LIN {X 0,Y 524.002,Z 47.209,A -85,B 0,C 180,E1 -4851.516,E2 -4851.516} C_VEL
LIN {X 0,Y 524.079,Z 47.2,A -85,B 0,C 180,E1 -4854.614,E2 -4854.614} C_VEL
LIN {X 0,Y 524.108,Z 47.2,A -85,B 0,C 180,E1 -4857.695,E2 -4857.695} C_VEL
LIN {X 0,Y 524.12,Z 47.194,A -85,B 0,C 180,E1 -4860.768,E2 -4860.768} C_VEL
LIN {X 0,Y 524.069,Z 47.199,A -85,B 0,C 180,E1 -4863.075,E2 -4863.075} C_VEL
LIN {X 0,Y 524.033,Z 47.205,A -85,B 0,C 180,E1 -4866.159,E2 -4866.159} C_VEL
LIN {X 0,Y 523.99,Z 47.215,A -85,B 0,C 180,E1 -4869.262,E2 -4869.262} C_VEL
LIN {X 0,Y 524.001,Z 47.209,A -85,B 0,C 180,E1 -4871.74,E2 -4871.74} C_VEL
LIN {X 0,Y 523.991,Z 47.217,A -85,B 0,C 180,E1 -4875.053,E2 -4875.053} C_VEL
LIN {X 0,Y 523.945,Z 47.214,A -85,B 0,C 180,E1 -4877.97,E2 -4877.97} C_VEL
LIN {X 0,Y 523.97,Z 47.215,A -85,B 0,C 180,E1 -4880.41,E2 -4880.41} C_VEL
LIN {X 0,Y 523.909,Z 47.228,A -85,B 0,C 180,E1 -4882.894,E2 -4882.894} C_VEL
LIN {X 0,Y 523.933,Z 47.216,A -85,B 0,C 180,E1 -4885.42,E2 -4885.42} C_VEL
LIN {X 0,Y 523.916,Z 47.222,A -85,B 0,C 180,E1 -4888.002,E2 -4888.002} C_VEL
LIN {X 0,Y 523.943,Z 47.219,A -85,B 0,C 180,E1 -4890.855,E2 -4890.855} C_VEL
LIN {X 0,Y 523.929,Z 47.219,A -85,B 0,C 180,E1 -4893.73,E2 -4893.73} C_VEL
LIN {X 0,Y 523.897,Z 47.228,A -85,B 0,C 180,E1 -4896.401,E2 -4896.401} C_VEL
LIN {X 0,Y 523.913,Z 47.221,A -85,B 0,C 180,E1 -4899.086,E2 -4899.086} C_VEL
LIN {X 0,Y 523.908,Z 47.229,A -85,B 0,C 180,E1 -4902.124,E2 -4902.124} C_VEL
LIN {X 0,Y 523.936,Z 47.219,A -85,B 0,C 180,E1 -4905.312,E2 -4905.312} C_VEL
LIN {X 0,Y 523.886,Z 47.226,A -85,B 0,C 180,E1 -4906.905,E2 -4906.905} C_VEL
LIN {X 0,Y 523.21,Z 47.316,A -85,B 0,C 180,E1 -4907.547,E2 -4907.547} C_VEL
LIN {X 0,Y 520.363,Z 47.669,A -85,B 0,C 180,E1 -4908.589,E2 -4908.589} C_VEL
LIN {X 0,Y 517.965,Z 47.967,A -85,B 0,C 180,E1 -4909.428,E2 -4909.428} C_VEL
LIN {X 0,Y 516.94,Z 48.093,A -85,B 0,C 180,E1 -4910.075,E2 -4910.075} C_VEL
LIN {X 0,Y 516.858,Z 48.101,A -85,B 0,C 180,E1 -4910.295,E2 -4910.295} C_VEL
LIN {X 0,Y 516.847,Z 48.108,A -85,B 0,C 180,E1 -4913.348,E2 -4913.348} C_VEL
LIN {X 0,Y 516.885,Z 48.101,A -85,B 0,C 180,E1 -4916.119,E2 -4916.119} C_VEL
LIN {X 0,Y 516.927,Z 48.11,A -85,B 0,C 180,E1 -4917.452,E2 -4917.452} C_VEL
LIN {X 0,Y 517.551,Z 52.851,A -85,B 0,C 180,E1 -4918.468,E2 -4918.468} C_VEL
LIN {X 0,Y 517.344,Z 63.831,A -85,B 0,C 180,E1 -4920.702,E2 -4920.702} C_VEL
LIN {X 0,Y 519.204,Z 73.107,A -85,B 0,C 180,E1 -4920.893,E2 -4920.893} C_VEL
LIN {X 0,Y 518.694,Z 170.265,A -85,B 0,C 180,E1 -4922.268,E2 -4922.268} C_VEL
LIN {X 0,Y 518.537,Z 183.805,A -85,B 0,C 180,E1 -4922.629,E2 -4922.629} C_VEL
LIN {X 0,Y 518.349,Z 195.673,A -85,B 0,C 180,E1 -4923.095,E2 -4923.095} C_VEL
LIN {X 0,Y 518.091,Z 206.71,A -85,B 0,C 180,E1 -4923.672,E2 -4923.672} C_VEL
LIN {X 0,Y 517.742,Z 217.113,A -85,B 0,C 180,E1 -4924.363,E2 -4924.363} C_VEL
LIN {X 0,Y 517.506,Z 227.582,A -85,B 0,C 180,E1 -4925.233,E2 -4925.233} C_VEL
LIN {X 0,Y 517.214,Z 236.66,A -85,B 0,C 180,E1 -4926.156,E2 -4926.156} C_VEL
LIN {X 0,Y 516.965,Z 245.113,A -85,B 0,C 180,E1 -4927.205,E2 -4927.205} C_VEL
LIN {X 0,Y 516.759,Z 252.003,A -85,B 0,C 180,E1 -4928.247,E2 -4928.247} C_VEL
LIN {X 0,Y 516.633,Z 257.643,A -85,B 0,C 180,E1 -4929.287,E2 -4929.287} C_VEL
LIN {X 0,Y 516.506,Z 263.065,A -85,B 0,C 180,E1 -4930.527,E2 -4930.527} C_VEL
LIN {X 0,Y 516.388,Z 267.182,A -85,B 0,C 180,E1 -4931.759,E2 -4931.759} C_VEL
LIN {X 0,Y 516.329,Z 269.267,A -85,B 0,C 180,E1 -4932.576,E2 -4932.576} C_VEL
LIN {X 0,Y 516.244,Z 270.907,A -85,B 0,C 180,E1 -4933.388,E2 -4933.388} C_VEL
LIN {X 0,Y 516.251,Z 272.102,A -85,B 0,C 180,E1 -4934.201,E2 -4934.201} C_VEL
LIN {X 0,Y 516.255,Z 272.907,A -85,B 0,C 180,E1 -4935.142,E2 -4935.142} C_VEL
LIN {X 0,Y 516.244,Z 273.078,A -85,B 0,C 180,E1 -4936.619,E2 -4936.619} C_VEL
LIN {X 0,Y 516.286,Z 272.561,A -85,B 0,C 180,E1 -4937.42,E2 -4937.42} C_VEL
LIN {X 0,Y 516.347,Z 271.191,A -85,B 0,C 180,E1 -4938.522,E2 -4938.522} C_VEL
LIN {X 0,Y 516.41,Z 267.483,A -85,B 0,C 180,E1 -4940.206,E2 -4940.206} C_VEL
LIN {X 0,Y 516.456,Z 263.649,A -85,B 0,C 180,E1 -4941.391,E2 -4941.391} C_VEL
LIN {X 0,Y 516.57,Z 258.69,A -85,B 0,C 180,E1 -4942.574,E2 -4942.574} C_VEL
LIN {X 0,Y 516.716,Z 252.475,A -85,B 0,C 180,E1 -4943.754,E2 -4943.754} C_VEL
LIN {X 0,Y 516.94,Z 244.707,A -85,B 0,C 180,E1 -4944.93,E2 -4944.93} C_VEL
LIN {X 0,Y 517.232,Z 235.046,A -85,B 0,C 180,E1 -4946.105,E2 -4946.105} C_VEL
LIN {X 0,Y 517.561,Z 225.026,A -85,B 0,C 180,E1 -4947.081,E2 -4947.081} C_VEL
LIN {X 0,Y 517.844,Z 215.126,A -85,B 0,C 180,E1 -4947.861,E2 -4947.861} C_VEL
LIN {X 0,Y 518.167,Z 202.649,A -85,B 0,C 180,E1 -4948.64,E2 -4948.64} C_VEL
LIN {X 0,Y 518.388,Z 190.252,A -85,B 0,C 180,E1 -4949.223,E2 -4949.223} C_VEL
LIN {X 0,Y 518.574,Z 177.905,A -85,B 0,C 180,E1 -4949.636,E2 -4949.636} C_VEL
LIN {X 0,Y 518.709,Z 165.439,A -85,B 0,C 180,E1 -4949.903,E2 -4949.903} C_VEL
LIN {X 0,Y 519.042,Z 71.979,A -85,B 0,C 180,E1 -4951.213,E2 -4951.213} C_VEL
LIN {X 0,Y 517.23,Z 63.405,A -85,B 0,C 180,E1 -4951.411,E2 -4951.411} C_VEL
LIN {X 0,Y 517.526,Z 53.185,A -85,B 0,C 180,E1 -4953.504,E2 -4953.504} C_VEL
LIN {X 0,Y 516.921,Z 48.099,A -85,B 0,C 180,E1 -4954.582,E2 -4954.582} C_VEL
LIN {X 0,Y 517.009,Z 48.085,A -85,B 0,C 180,E1 -4957.096,E2 -4957.096} C_VEL
LIN {X 0,Y 516.95,Z 48.087,A -85,B 0,C 180,E1 -4959.39,E2 -4959.39} C_VEL
LIN {X 0,Y 516.958,Z 48.086,A -85,B 0,C 180,E1 -4961.807,E2 -4961.807} C_VEL
LIN {X 0,Y 516.951,Z 48.087,A -85,B 0,C 180,E1 -4965.147,E2 -4965.147} C_VEL
LIN {X 0,Y 516.922,Z 48.098,A -85,B 0,C 180,E1 -4968.223,E2 -4968.223} C_VEL
LIN {X 0,Y 516.918,Z 48.093,A -85,B 0,C 180,E1 -4970.701,E2 -4970.701} C_VEL
LIN {X 0,Y 516.897,Z 48.102,A -85,B 0,C 180,E1 -4974.073,E2 -4974.073} C_VEL
LIN {X 0,Y 516.931,Z 48.09,A -85,B 0,C 180,E1 -4976.658,E2 -4976.658} C_VEL
LIN {X 0,Y 516.916,Z 48.094,A -85,B 0,C 180,E1 -4979.523,E2 -4979.523} C_VEL
LIN {X 0,Y 516.901,Z 48.093,A -85,B 0,C 180,E1 -4982.543,E2 -4982.543} C_VEL
LIN {X 0,Y 516.885,Z 48.098,A -85,B 0,C 180,E1 -4985.332,E2 -4985.332} C_VEL
LIN {X 0,Y 516.885,Z 48.099,A -85,B 0,C 180,E1 -4987.943,E2 -4987.943} C_VEL
LIN {X 0,Y 516.887,Z 48.095,A -85,B 0,C 180,E1 -4990.742,E2 -4990.742} C_VEL
LIN {X 0,Y 516.887,Z 48.096,A -85,B 0,C 180,E1 -4992.831,E2 -4992.831} C_VEL
LIN {X 0,Y 516.899,Z 48.097,A -85,B 0,C 180,E1 -4995.007,E2 -4995.007} C_VEL
LIN {X 0,Y 516.917,Z 48.091,A -85,B 0,C 180,E1 -4998.399,E2 -4998.399} C_VEL
LIN {X 0,Y 516.886,Z 48.101,A -85,B 0,C 180,E1 -5001.284,E2 -5001.284} C_VEL
LIN {X 0,Y 516.875,Z 48.096,A -85,B 0,C 180,E1 -5004.22,E2 -5004.22} C_VEL
LIN {X 0,Y 516.898,Z 48.1,A -85,B 0,C 180,E1 -5007.053,E2 -5007.053} C_VEL
LIN {X 0,Y 516.896,Z 48.093,A -85,B 0,C 180,E1 -5009.796,E2 -5009.796} C_VEL
LIN {X 0,Y 516.93,Z 48.094,A -85,B 0,C 180,E1 -5012.467,E2 -5012.467} C_VEL
LIN {X 0,Y 516.914,Z 48.094,A -85,B 0,C 180,E1 -5015.072,E2 -5015.072} C_VEL
LIN {X 0,Y 516.89,Z 48.102,A -85,B 0,C 180,E1 -5018.462,E2 -5018.462} C_VEL
LIN {X 0,Y 516.904,Z 48.095,A -85,B 0,C 180,E1 -5020.955,E2 -5020.955} C_VEL
LIN {X 0,Y 516.916,Z 48.091,A -85,B 0,C 180,E1 -5023.41,E2 -5023.41} C_VEL
LIN {X 0,Y 516.897,Z 48.096,A -85,B 0,C 180,E1 -5025.833,E2 -5025.833} C_VEL
LIN {X 0,Y 516.969,Z 48.093,A -85,B 0,C 180,E1 -5028.233,E2 -5028.233} C_VEL
LIN {X 0,Y 516.968,Z 48.085,A -85,B 0,C 180,E1 -5031.399,E2 -5031.399} C_VEL
LIN {X 0,Y 517.011,Z 48.084,A -85,B 0,C 180,E1 -5033.757,E2 -5033.757} C_VEL
LIN {X 0,Y 517.084,Z 48.076,A -85,B 0,C 180,E1 -5037.663,E2 -5037.663} C_VEL
LIN {X 0,Y 517.094,Z 48.069,A -85,B 0,C 180,E1 -5040.779,E2 -5040.779} C_VEL
LIN {X 0,Y 517.012,Z 48.081,A -85,B 0,C 180,E1 -5043.117,E2 -5043.117} C_VEL
LIN {X 0,Y 517.003,Z 48.081,A -85,B 0,C 180,E1 -5046.243,E2 -5046.243} C_VEL
LIN {X 0,Y 516.949,Z 48.095,A -85,B 0,C 180,E1 -5049.389,E2 -5049.389} C_VEL
LIN {X 0,Y 516.954,Z 48.089,A -85,B 0,C 180,E1 -5051.807,E2 -5051.807} C_VEL
LIN {X 0,Y 516.947,Z 48.094,A -85,B 0,C 180,E1 -5055.146,E2 -5055.146} C_VEL
LIN {X 0,Y 516.918,Z 48.091,A -85,B 0,C 180,E1 -5058.222,E2 -5058.222} C_VEL
LIN {X 0,Y 516.914,Z 48.095,A -85,B 0,C 180,E1 -5060.701,E2 -5060.701} C_VEL
LIN {X 0,Y 516.904,Z 48.092,A -85,B 0,C 180,E1 -5064.072,E2 -5064.072} C_VEL
LIN {X 0,Y 516.906,Z 48.098,A -85,B 0,C 180,E1 -5066.659,E2 -5066.659} C_VEL
LIN {X 0,Y 516.913,Z 48.092,A -85,B 0,C 180,E1 -5069.524,E2 -5069.524} C_VEL
LIN {X 0,Y 516.897,Z 48.101,A -85,B 0,C 180,E1 -5072.543,E2 -5072.543} C_VEL
LIN {X 0,Y 516.868,Z 48.097,A -85,B 0,C 180,E1 -5075.33,E2 -5075.33} C_VEL
LIN {X 0,Y 516.882,Z 48.097,A -85,B 0,C 180,E1 -5077.943,E2 -5077.943} C_VEL
LIN {X 0,Y 516.885,Z 48.098,A -85,B 0,C 180,E1 -5080.742,E2 -5080.742} C_VEL
LIN {X 0,Y 516.884,Z 48.097,A -85,B 0,C 180,E1 -5082.831,E2 -5082.831} C_VEL
LIN {X 0,Y 516.897,Z 48.094,A -85,B 0,C 180,E1 -5085.007,E2 -5085.007} C_VEL
LIN {X 0,Y 516.915,Z 48.095,A -85,B 0,C 180,E1 -5088.399,E2 -5088.399} C_VEL
LIN {X 0,Y 516.882,Z 48.096,A -85,B 0,C 180,E1 -5091.284,E2 -5091.284} C_VEL
LIN {X 0,Y 516.873,Z 48.1,A -85,B 0,C 180,E1 -5094.22,E2 -5094.22} C_VEL
LIN {X 0,Y 516.897,Z 48.094,A -85,B 0,C 180,E1 -5097.053,E2 -5097.053} C_VEL
LIN {X 0,Y 516.89,Z 48.103,A -85,B 0,C 180,E1 -5099.796,E2 -5099.796} C_VEL
LIN {X 0,Y 516.928,Z 48.093,A -85,B 0,C 180,E1 -5102.467,E2 -5102.467} C_VEL
LIN {X 0,Y 516.966,Z 48.155,A -85,B 0,C 180,E1 -5104.536,E2 -5104.536} C_VEL
LIN {X 0,Y 518.452,Z 56.246,A -85,B 0,C 180,E1 -5105.834,E2 -5105.834} C_VEL
LIN {X 0,Y 518.155,Z 71.32,A -85,B 0,C 180,E1 -5108.099,E2 -5108.099} C_VEL
LIN {X 0,Y 517.783,Z 88.007,A -85,B 0,C 180,E1 -5110.576,E2 -5110.576} C_VEL
LIN {X 0,Y 517.364,Z 107.405,A -85,B 0,C 180,E1 -5113.425,E2 -5113.425} C_VEL
LIN {X 0,Y 517.194,Z 115.539,A -85,B 0,C 180,E1 -5114.611,E2 -5114.611} C_VEL
LIN {X 0,Y 519.007,Z 128.795,A -85,B 0,C 180,E1 -5114.864,E2 -5114.864} C_VEL
LIN {X 0,Y 518.582,Z 224.127,A -85,B 0,C 180,E1 -5116.205,E2 -5116.205} C_VEL
LIN {X 0,Y 518.303,Z 237.516,A -85,B 0,C 180,E1 -5116.548,E2 -5116.548} C_VEL
LIN {X 0,Y 518.035,Z 249.752,A -85,B 0,C 180,E1 -5117.015,E2 -5117.015} C_VEL
LIN {X 0,Y 517.755,Z 261.479,A -85,B 0,C 180,E1 -5117.617,E2 -5117.617} C_VEL
LIN {X 0,Y 517.449,Z 272.455,A -85,B 0,C 180,E1 -5118.344,E2 -5118.344} C_VEL
LIN {X 0,Y 517.167,Z 283.173,A -85,B 0,C 180,E1 -5119.23,E2 -5119.23} C_VEL
LIN {X 0,Y 516.841,Z 292.831,A -85,B 0,C 180,E1 -5120.213,E2 -5120.213} C_VEL
LIN {X 0,Y 516.653,Z 300.756,A -85,B 0,C 180,E1 -5121.197,E2 -5121.197} C_VEL
LIN {X 0,Y 516.502,Z 308.499,A -85,B 0,C 180,E1 -5122.376,E2 -5122.376} C_VEL
LIN {X 0,Y 516.353,Z 315.634,A -85,B 0,C 180,E1 -5123.749,E2 -5123.749} C_VEL
LIN {X 0,Y 516.311,Z 320.385,A -85,B 0,C 180,E1 -5124.924,E2 -5124.924} C_VEL
LIN {X 0,Y 516.369,Z 324.019,A -85,B 0,C 180,E1 -5126.098,E2 -5126.098} C_VEL
LIN {X 0,Y 516.326,Z 325.889,A -85,B 0,C 180,E1 -5126.879,E2 -5126.879} C_VEL
LIN {X 0,Y 516.266,Z 327.29,A -85,B 0,C 180,E1 -5127.659,E2 -5127.659} C_VEL
LIN {X 0,Y 516.189,Z 328.896,A -85,B 0,C 180,E1 -5129.22,E2 -5129.22} C_VEL
LIN {X 0,Y 516.194,Z 329.111,A -85,B 0,C 180,E1 -5130,E2 -5130} C_VEL
LIN {X 0,Y 516.189,Z 328.891,A -85,B 0,C 180,E1 -5130.78,E2 -5130.78} C_VEL
LIN {X 0,Y 516.266,Z 327.277,A -85,B 0,C 180,E1 -5132.34,E2 -5132.34} C_VEL
LIN {X 0,Y 516.326,Z 325.873,A -85,B 0,C 180,E1 -5133.121,E2 -5133.121} C_VEL
LIN {X 0,Y 516.311,Z 322.912,A -85,B 0,C 180,E1 -5134.293,E2 -5134.293} C_VEL
LIN {X 0,Y 516.363,Z 318.91,A -85,B 0,C 180,E1 -5135.467,E2 -5135.467} C_VEL
LIN {X 0,Y 516.405,Z 313.108,A -85,B 0,C 180,E1 -5136.771,E2 -5136.771} C_VEL
LIN {X 0,Y 516.557,Z 306.034,A -85,B 0,C 180,E1 -5138.016,E2 -5138.016} C_VEL
LIN {X 0,Y 516.723,Z 297.697,A -85,B 0,C 180,E1 -5139.196,E2 -5139.196} C_VEL
LIN {X 0,Y 516.941,Z 289.155,A -85,B 0,C 180,E1 -5140.18,E2 -5140.18} C_VEL
LIN {X 0,Y 517.281,Z 278.611,A -85,B 0,C 180,E1 -5141.163,E2 -5141.163} C_VEL
LIN {X 0,Y 517.565,Z 266.99,A -85,B 0,C 180,E1 -5142.033,E2 -5142.033} C_VEL
LIN {X 0,Y 517.952,Z 254.814,A -85,B 0,C 180,E1 -5142.738,E2 -5142.738} C_VEL
LIN {X 0,Y 518.157,Z 243.707,A -85,B 0,C 180,E1 -5143.231,E2 -5143.231} C_VEL
LIN {X 0,Y 518.419,Z 230.576,A -85,B 0,C 180,E1 -5143.648,E2 -5143.648} C_VEL
LIN {X 0,Y 518.65,Z 218.043,A -85,B 0,C 180,E1 -5143.892,E2 -5143.892} C_VEL
LIN {X 0,Y 518.952,Z 128.16,A -85,B 0,C 180,E1 -5145.145,E2 -5145.145} C_VEL
LIN {X 0,Y 517.214,Z 115.433,A -85,B 0,C 180,E1 -5145.384,E2 -5145.384} C_VEL
LIN {X 0,Y 517.715,Z 92.05,A -85,B 0,C 180,E1 -5148.808,E2 -5148.808} C_VEL
LIN {X 0,Y 518.116,Z 72.687,A -85,B 0,C 180,E1 -5151.693,E2 -5151.693} C_VEL
LIN {X 0,Y 518.514,Z 56.387,A -85,B 0,C 180,E1 -5154.161,E2 -5154.161} C_VEL
LIN {X 0,Y 516.943,Z 48.093,A -85,B 0,C 180,E1 -5155.545,E2 -5155.545} C_VEL
LIN {X 0,Y 516.92,Z 48.099,A -85,B 0,C 180,E1 -5158.415,E2 -5158.415} C_VEL
LIN {X 0,Y 516.889,Z 48.098,A -85,B 0,C 180,E1 -5161.109,E2 -5161.109} C_VEL
LIN {X 0,Y 516.891,Z 48.103,A -85,B 0,C 180,E1 -5163.963,E2 -5163.963} C_VEL
LIN {X 0,Y 516.883,Z 48.097,A -85,B 0,C 180,E1 -5166.745,E2 -5166.745} C_VEL
LIN {X 0,Y 516.881,Z 48.103,A -85,B 0,C 180,E1 -5169.721,E2 -5169.721} C_VEL
LIN {X 0,Y 516.91,Z 48.1,A -85,B 0,C 180,E1 -5171.775,E2 -5171.775} C_VEL
LIN {X 0,Y 516.893,Z 48.094,A -85,B 0,C 180,E1 -5175.007,E2 -5175.007} C_VEL
LIN {X 0,Y 516.921,Z 48.091,A -85,B 0,C 180,E1 -5178.397,E2 -5178.397} C_VEL
LIN {X 0,Y 516.885,Z 48.103,A -85,B 0,C 180,E1 -5181.284,E2 -5181.284} C_VEL
LIN {X 0,Y 516.89,Z 48.095,A -85,B 0,C 180,E1 -5184.221,E2 -5184.221} C_VEL
LIN {X 0,Y 516.894,Z 48.101,A -85,B 0,C 180,E1 -5187.053,E2 -5187.053} C_VEL
LIN {X 0,Y 516.89,Z 48.094,A -85,B 0,C 180,E1 -5189.796,E2 -5189.796} C_VEL
LIN {X 0,Y 516.926,Z 48.093,A -85,B 0,C 180,E1 -5192.467,E2 -5192.467} C_VEL
LIN {X 0,Y 516.909,Z 48.097,A -85,B 0,C 180,E1 -5195.072,E2 -5195.072} C_VEL
LIN {X 0,Y 516.867,Z 48.094,A -85,B 0,C 180,E1 -5197.621,E2 -5197.621} C_VEL
LIN {X 0,Y 516.93,Z 48.092,A -85,B 0,C 180,E1 -5200.13,E2 -5200.13} C_VEL
LIN {X 0,Y 516.927,Z 48.095,A -85,B 0,C 180,E1 -5202.596,E2 -5202.596} C_VEL
LIN {X 0,Y 516.94,Z 48.089,A -85,B 0,C 180,E1 -5205.03,E2 -5205.03} C_VEL
LIN {X 0,Y 516.963,Z 48.09,A -85,B 0,C 180,E1 -5208.234,E2 -5208.234} C_VEL
LIN {X 0,Y 516.967,Z 48.085,A -85,B 0,C 180,E1 -5211.4,E2 -5211.4} C_VEL
LIN {X 0,Y 517.007,Z 48.083,A -85,B 0,C 180,E1 -5213.757,E2 -5213.757} C_VEL
LIN {X 0,Y 517.08,Z 48.075,A -85,B 0,C 180,E1 -5217.663,E2 -5217.663} C_VEL
LIN {X 0,Y 517.091,Z 48.07,A -85,B 0,C 180,E1 -5220.779,E2 -5220.779} C_VEL
LIN {X 0,Y 517.009,Z 48.079,A -85,B 0,C 180,E1 -5223.117,E2 -5223.117} C_VEL
LIN {X 0,Y 516.999,Z 48.081,A -85,B 0,C 180,E1 -5226.244,E2 -5226.244} C_VEL
LIN {X 0,Y 516.946,Z 48.094,A -85,B 0,C 180,E1 -5229.39,E2 -5229.39} C_VEL
LIN {X 0,Y 516.95,Z 48.087,A -85,B 0,C 180,E1 -5231.807,E2 -5231.807} C_VEL
LIN {X 0,Y 516.943,Z 48.096,A -85,B 0,C 180,E1 -5235.147,E2 -5235.147} C_VEL
LIN {X 0,Y 516.914,Z 48.09,A -85,B 0,C 180,E1 -5238.223,E2 -5238.223} C_VEL
LIN {X 0,Y 516.911,Z 48.099,A -85,B 0,C 180,E1 -5240.702,E2 -5240.702} C_VEL
LIN {X 0,Y 516.9,Z 48.095,A -85,B 0,C 180,E1 -5244.073,E2 -5244.073} C_VEL
LIN {X 0,Y 516.896,Z 48.101,A -85,B 0,C 180,E1 -5246.66,E2 -5246.66} C_VEL
LIN {X 0,Y 516.909,Z 48.091,A -85,B 0,C 180,E1 -5249.524,E2 -5249.524} C_VEL
LIN {X 0,Y 516.893,Z 48.1,A -85,B 0,C 180,E1 -5252.544,E2 -5252.544} C_VEL
LIN {X 0,Y 516.861,Z 48.097,A -85,B 0,C 180,E1 -5255.329,E2 -5255.329} C_VEL
LIN {X 0,Y 516.878,Z 48.103,A -85,B 0,C 180,E1 -5257.943,E2 -5257.943} C_VEL
LIN {X 0,Y 516.853,Z 48.097,A -85,B 0,C 180,E1 -5260.745,E2 -5260.745} C_VEL
LIN {X 0,Y 516.88,Z 48.104,A -85,B 0,C 180,E1 -5263.904,E2 -5263.904} C_VEL
LIN {X 0,Y 516.84,Z 48.104,A -85,B 0,C 180,E1 -5266.906,E2 -5266.906} C_VEL
LIN {X 0,Y 516.861,Z 48.107,A -85,B 0,C 180,E1 -5269.594,E2 -5269.594} C_VEL
LIN {X 0,Y 516.858,Z 48.101,A -85,B 0,C 180,E1 -5270.295,E2 -5270.295} C_VEL
LIN {X 0,Y 516.196,Z 48.184,A -85,B 0,C 180,E1 -5270.945,E2 -5270.945} C_VEL
LIN {X 0,Y 513.345,Z 48.545,A -85,B 0,C 180,E1 -5272,E2 -5272} C_VEL
LIN {X 0,Y 510.929,Z 48.849,A -85,B 0,C 180,E1 -5272.851,E2 -5272.851} C_VEL
LIN {X 0,Y 509.888,Z 48.976,A -85,B 0,C 180,E1 -5273.507,E2 -5273.507} C_VEL
LIN {X 0,Y 509.802,Z 48.985,A -85,B 0,C 180,E1 -5273.73,E2 -5273.73} C_VEL
LIN {X 0,Y 509.849,Z 48.978,A -85,B 0,C 180,E1 -5276.539,E2 -5276.539} C_VEL
LIN {X 0,Y 509.91,Z 49.086,A -85,B 0,C 180,E1 -5277.322,E2 -5277.322} C_VEL
LIN {X 0,Y 510.594,Z 54.905,A -85,B 0,C 180,E1 -5278.583,E2 -5278.583} C_VEL
LIN {X 0,Y 510.368,Z 64.136,A -85,B 0,C 180,E1 -5280.478,E2 -5280.478} C_VEL
LIN {X 0,Y 512.376,Z 74.317,A -85,B 0,C 180,E1 -5280.692,E2 -5280.692} C_VEL
LIN {X 0,Y 511.822,Z 170.404,A -85,B 0,C 180,E1 -5282.071,E2 -5282.071} C_VEL
LIN {X 0,Y 511.635,Z 184.046,A -85,B 0,C 180,E1 -5282.436,E2 -5282.436} C_VEL
LIN {X 0,Y 511.442,Z 196.255,A -85,B 0,C 180,E1 -5282.923,E2 -5282.923} C_VEL
LIN {X 0,Y 511.12,Z 208.288,A -85,B 0,C 180,E1 -5283.574,E2 -5283.574} C_VEL
LIN {X 0,Y 510.759,Z 218.975,A -85,B 0,C 180,E1 -5284.315,E2 -5284.315} C_VEL
LIN {X 0,Y 510.464,Z 229.831,A -85,B 0,C 180,E1 -5285.257,E2 -5285.257} C_VEL
LIN {X 0,Y 510.17,Z 238.963,A -85,B 0,C 180,E1 -5286.238,E2 -5286.238} C_VEL
LIN {X 0,Y 509.869,Z 248.021,A -85,B 0,C 180,E1 -5287.448,E2 -5287.448} C_VEL
LIN {X 0,Y 509.653,Z 254.798,A -85,B 0,C 180,E1 -5288.566,E2 -5288.566} C_VEL
LIN {X 0,Y 509.519,Z 260.942,A -85,B 0,C 180,E1 -5289.829,E2 -5289.829} C_VEL
LIN {X 0,Y 509.36,Z 265.677,A -85,B 0,C 180,E1 -5291.08,E2 -5291.08} C_VEL
LIN {X 0,Y 509.273,Z 269.205,A -85,B 0,C 180,E1 -5292.326,E2 -5292.326} C_VEL
LIN {X 0,Y 509.196,Z 270.929,A -85,B 0,C 180,E1 -5293.152,E2 -5293.152} C_VEL
LIN {X 0,Y 509.178,Z 272.225,A -85,B 0,C 180,E1 -5293.976,E2 -5293.976} C_VEL
LIN {X 0,Y 509.176,Z 273.25,A -85,B 0,C 180,E1 -5295.06,E2 -5295.06} C_VEL
LIN {X 0,Y 509.149,Z 273.502,A -85,B 0,C 180,E1 -5296.429,E2 -5296.429} C_VEL
LIN {X 0,Y 509.189,Z 273.11,A -85,B 0,C 180,E1 -5297.242,E2 -5297.242} C_VEL
LIN {X 0,Y 509.257,Z 271.687,A -85,B 0,C 180,E1 -5298.477,E2 -5298.477} C_VEL
LIN {X 0,Y 509.313,Z 268.385,A -85,B 0,C 180,E1 -5300.068,E2 -5300.068} C_VEL
LIN {X 0,Y 509.387,Z 264.72,A -85,B 0,C 180,E1 -5301.271,E2 -5301.271} C_VEL
LIN {X 0,Y 509.495,Z 259.945,A -85,B 0,C 180,E1 -5302.47,E2 -5302.47} C_VEL
LIN {X 0,Y 509.672,Z 252.821,A -85,B 0,C 180,E1 -5303.866,E2 -5303.866} C_VEL
LIN {X 0,Y 509.923,Z 245.037,A -85,B 0,C 180,E1 -5305.059,E2 -5305.059} C_VEL
LIN {X 0,Y 510.246,Z 235.36,A -85,B 0,C 180,E1 -5306.249,E2 -5306.249} C_VEL
LIN {X 0,Y 510.595,Z 225.316,A -85,B 0,C 180,E1 -5307.239,E2 -5307.239} C_VEL
LIN {X 0,Y 510.915,Z 215.385,A -85,B 0,C 180,E1 -5308.03,E2 -5308.03} C_VEL
LIN {X 0,Y 511.224,Z 204.606,A -85,B 0,C 180,E1 -5308.72,E2 -5308.72} C_VEL
LIN {X 0,Y 511.454,Z 192.762,A -85,B 0,C 180,E1 -5309.311,E2 -5309.311} C_VEL
LIN {X 0,Y 511.676,Z 180.616,A -85,B 0,C 180,E1 -5309.754,E2 -5309.754} C_VEL
LIN {X 0,Y 511.819,Z 168.222,A -85,B 0,C 180,E1 -5310.049,E2 -5310.049} C_VEL
LIN {X 0,Y 512.176,Z 72.822,A -85,B 0,C 180,E1 -5311.41,E2 -5311.41} C_VEL
LIN {X 0,Y 510.272,Z 63.821,A -85,B 0,C 180,E1 -5311.603,E2 -5311.603} C_VEL
LIN {X 0,Y 510.462,Z 52.48,A -85,B 0,C 180,E1 -5313.948,E2 -5313.948} C_VEL
LIN {X 0,Y 509.906,Z 48.973,A -85,B 0,C 180,E1 -5314.744,E2 -5314.744} C_VEL
LIN {X 0,Y 509.981,Z 48.96,A -85,B 0,C 180,E1 -5317.145,E2 -5317.145} C_VEL
LIN {X 0,Y 509.861,Z 48.975,A -85,B 0,C 180,E1 -5320.323,E2 -5320.323} C_VEL
LIN {X 0,Y 509.883,Z 48.972,A -85,B 0,C 180,E1 -5322.741,E2 -5322.741} C_VEL
LIN {X 0,Y 509.9,Z 48.965,A -85,B 0,C 180,E1 -5325.242,E2 -5325.242} C_VEL
LIN {X 0,Y 509.867,Z 48.975,A -85,B 0,C 180,E1 -5328.484,E2 -5328.484} C_VEL
LIN {X 0,Y 509.856,Z 48.971,A -85,B 0,C 180,E1 -5331.002,E2 -5331.002} C_VEL
LIN {X 0,Y 509.828,Z 48.976,A -85,B 0,C 180,E1 -5333.564,E2 -5333.564} C_VEL
LIN {X 0,Y 509.917,Z 48.966,A -85,B 0,C 180,E1 -5336.378,E2 -5336.378} C_VEL
LIN {X 0,Y 509.878,Z 48.968,A -85,B 0,C 180,E1 -5338.844,E2 -5338.844} C_VEL
LIN {X 0,Y 509.826,Z 48.979,A -85,B 0,C 180,E1 -5341.59,E2 -5341.59} C_VEL
LIN {X 0,Y 509.858,Z 48.971,A -85,B 0,C 180,E1 -5344.413,E2 -5344.413} C_VEL
LIN {X 0,Y 509.823,Z 48.979,A -85,B 0,C 180,E1 -5347.341,E2 -5347.341} C_VEL
LIN {X 0,Y 509.843,Z 48.972,A -85,B 0,C 180,E1 -5350.382,E2 -5350.382} C_VEL
LIN {X 0,Y 509.827,Z 48.977,A -85,B 0,C 180,E1 -5353.062,E2 -5353.062} C_VEL
LIN {X 0,Y 509.826,Z 48.977,A -85,B 0,C 180,E1 -5355.793,E2 -5355.793} C_VEL
LIN {X 0,Y 509.859,Z 48.971,A -85,B 0,C 180,E1 -5358.574,E2 -5358.574} C_VEL
LIN {X 0,Y 509.855,Z 48.972,A -85,B 0,C 180,E1 -5361.786,E2 -5361.786} C_VEL
LIN {X 0,Y 509.835,Z 48.976,A -85,B 0,C 180,E1 -5364.622,E2 -5364.622} C_VEL
LIN {X 0,Y 509.865,Z 48.971,A -85,B 0,C 180,E1 -5367.481,E2 -5367.481} C_VEL
LIN {X 0,Y 509.862,Z 48.971,A -85,B 0,C 180,E1 -5370.273,E2 -5370.273} C_VEL
LIN {X 0,Y 509.887,Z 48.972,A -85,B 0,C 180,E1 -5372.944,E2 -5372.944} C_VEL
LIN {X 0,Y 509.874,Z 48.968,A -85,B 0,C 180,E1 -5375.574,E2 -5375.574} C_VEL
LIN {X 0,Y 509.854,Z 48.973,A -85,B 0,C 180,E1 -5378.998,E2 -5378.998} C_VEL
LIN {X 0,Y 509.885,Z 48.97,A -85,B 0,C 180,E1 -5382.001,E2 -5382.001} C_VEL
LIN {X 0,Y 509.914,Z 48.965,A -85,B 0,C 180,E1 -5384.819,E2 -5384.819} C_VEL
LIN {X 0,Y 509.904,Z 48.972,A -85,B 0,C 180,E1 -5388.124,E2 -5388.124} C_VEL
LIN {X 0,Y 509.914,Z 48.963,A -85,B 0,C 180,E1 -5391.28,E2 -5391.28} C_VEL
LIN {X 0,Y 509.962,Z 48.961,A -85,B 0,C 180,E1 -5393.67,E2 -5393.67} C_VEL
LIN {X 0,Y 510.055,Z 48.951,A -85,B 0,C 180,E1 -5397.631,E2 -5397.631} C_VEL
LIN {X 0,Y 510.065,Z 48.944,A -85,B 0,C 180,E1 -5400.789,E2 -5400.789} C_VEL
LIN {X 0,Y 509.954,Z 48.96,A -85,B 0,C 180,E1 -5403.16,E2 -5403.16} C_VEL
LIN {X 0,Y 509.954,Z 48.959,A -85,B 0,C 180,E1 -5406.33,E2 -5406.33} C_VEL
LIN {X 0,Y 509.89,Z 48.974,A -85,B 0,C 180,E1 -5409.52,E2 -5409.52} C_VEL
LIN {X 0,Y 509.907,Z 48.966,A -85,B 0,C 180,E1 -5411.931,E2 -5411.931} C_VEL
LIN {X 0,Y 509.896,Z 48.974,A -85,B 0,C 180,E1 -5415.242,E2 -5415.242} C_VEL
LIN {X 0,Y 509.869,Z 48.969,A -85,B 0,C 180,E1 -5417.993,E2 -5417.993} C_VEL
LIN {X 0,Y 509.888,Z 48.967,A -85,B 0,C 180,E1 -5420.401,E2 -5420.401} C_VEL
LIN {X 0,Y 509.831,Z 48.975,A -85,B 0,C 180,E1 -5423.563,E2 -5423.563} C_VEL
LIN {X 0,Y 509.888,Z 48.969,A -85,B 0,C 180,E1 -5426.372,E2 -5426.372} C_VEL
LIN {X 0,Y 509.874,Z 48.976,A -85,B 0,C 180,E1 -5428.844,E2 -5428.844} C_VEL
LIN {X 0,Y 509.821,Z 48.975,A -85,B 0,C 180,E1 -5431.59,E2 -5431.59} C_VEL
LIN {X 0,Y 509.849,Z 48.977,A -85,B 0,C 180,E1 -5434.414,E2 -5434.414} C_VEL
LIN {X 0,Y 509.818,Z 48.975,A -85,B 0,C 180,E1 -5437.341,E2 -5437.341} C_VEL
LIN {X 0,Y 509.84,Z 48.981,A -85,B 0,C 180,E1 -5440.382,E2 -5440.382} C_VEL
LIN {X 0,Y 509.824,Z 48.975,A -85,B 0,C 180,E1 -5443.062,E2 -5443.062} C_VEL
LIN {X 0,Y 509.824,Z 48.978,A -85,B 0,C 180,E1 -5445.793,E2 -5445.793} C_VEL
LIN {X 0,Y 509.857,Z 48.972,A -85,B 0,C 180,E1 -5448.574,E2 -5448.574} C_VEL
LIN {X 0,Y 509.852,Z 48.977,A -85,B 0,C 180,E1 -5451.787,E2 -5451.787} C_VEL
LIN {X 0,Y 509.832,Z 48.974,A -85,B 0,C 180,E1 -5454.622,E2 -5454.622} C_VEL
LIN {X 0,Y 509.863,Z 48.974,A -85,B 0,C 180,E1 -5457.481,E2 -5457.481} C_VEL
LIN {X 0,Y 509.861,Z 48.976,A -85,B 0,C 180,E1 -5460.274,E2 -5460.274} C_VEL
LIN {X 0,Y 509.886,Z 48.972,A -85,B 0,C 180,E1 -5462.944,E2 -5462.944} C_VEL
LIN {X 0,Y 509.93,Z 49.078,A -85,B 0,C 180,E1 -5464.379,E2 -5464.379} C_VEL
LIN {X 0,Y 511.559,Z 58.313,A -85,B 0,C 180,E1 -5465.875,E2 -5465.875} C_VEL
LIN {X 0,Y 511.097,Z 77.853,A -85,B 0,C 180,E1 -5468.841,E2 -5468.841} C_VEL
LIN {X 0,Y 510.566,Z 100.441,A -85,B 0,C 180,E1 -5472.219,E2 -5472.219} C_VEL
LIN {X 0,Y 510.178,Z 115.221,A -85,B 0,C 180,E1 -5474.406,E2 -5474.406} C_VEL
LIN {X 0,Y 512.136,Z 129.771,A -85,B 0,C 180,E1 -5474.678,E2 -5474.678} C_VEL
LIN {X 0,Y 511.675,Z 224.809,A -85,B 0,C 180,E1 -5476.041,E2 -5476.041} C_VEL
LIN {X 0,Y 511.363,Z 237.843,A -85,B 0,C 180,E1 -5476.387,E2 -5476.387} C_VEL
LIN {X 0,Y 511.076,Z 250.467,A -85,B 0,C 180,E1 -5476.885,E2 -5476.885} C_VEL
LIN {X 0,Y 510.748,Z 262.481,A -85,B 0,C 180,E1 -5477.533,E2 -5477.533} C_VEL
LIN {X 0,Y 510.432,Z 273.362,A -85,B 0,C 180,E1 -5478.282,E2 -5478.282} C_VEL
LIN {X 0,Y 510.122,Z 283.86,A -85,B 0,C 180,E1 -5479.18,E2 -5479.18} C_VEL
LIN {X 0,Y 509.804,Z 292.443,A -85,B 0,C 180,E1 -5480.077,E2 -5480.077} C_VEL
LIN {X 0,Y 509.6,Z 300.369,A -85,B 0,C 180,E1 -5481.074,E2 -5481.074} C_VEL
LIN {X 0,Y 509.415,Z 308.113,A -85,B 0,C 180,E1 -5482.269,E2 -5482.269} C_VEL
LIN {X 0,Y 509.259,Z 315.249,A -85,B 0,C 180,E1 -5483.661,E2 -5483.661} C_VEL
LIN {X 0,Y 509.239,Z 320.002,A -85,B 0,C 180,E1 -5484.853,E2 -5484.853} C_VEL
LIN {X 0,Y 509.275,Z 323.635,A -85,B 0,C 180,E1 -5486.043,E2 -5486.043} C_VEL
LIN {X 0,Y 509.241,Z 325.506,A -85,B 0,C 180,E1 -5486.835,E2 -5486.835} C_VEL
LIN {X 0,Y 509.196,Z 326.908,A -85,B 0,C 180,E1 -5487.627,E2 -5487.627} C_VEL
LIN {X 0,Y 509.101,Z 328.512,A -85,B 0,C 180,E1 -5489.209,E2 -5489.209} C_VEL
LIN {X 0,Y 509.105,Z 328.727,A -85,B 0,C 180,E1 -5490,E2 -5490} C_VEL
LIN {X 0,Y 509.12,Z 327.893,A -85,B 0,C 180,E1 -5491.582,E2 -5491.582} C_VEL
LIN {X 0,Y 509.196,Z 326.892,A -85,B 0,C 180,E1 -5492.373,E2 -5492.373} C_VEL
LIN {X 0,Y 509.241,Z 325.485,A -85,B 0,C 180,E1 -5493.164,E2 -5493.164} C_VEL
LIN {X 0,Y 509.204,Z 322.522,A -85,B 0,C 180,E1 -5494.353,E2 -5494.353} C_VEL
LIN {X 0,Y 509.272,Z 318.518,A -85,B 0,C 180,E1 -5495.543,E2 -5495.543} C_VEL
LIN {X 0,Y 509.329,Z 312.462,A -85,B 0,C 180,E1 -5496.914,E2 -5496.914} C_VEL
LIN {X 0,Y 509.476,Z 305.636,A -85,B 0,C 180,E1 -5498.128,E2 -5498.128} C_VEL
LIN {X 0,Y 509.68,Z 297.298,A -85,B 0,C 180,E1 -5499.324,E2 -5499.324} C_VEL
LIN {X 0,Y 509.926,Z 288.754,A -85,B 0,C 180,E1 -5500.321,E2 -5500.321} C_VEL
LIN {X 0,Y 510.291,Z 278.212,A -85,B 0,C 180,E1 -5501.318,E2 -5501.318} C_VEL
LIN {X 0,Y 510.565,Z 267.349,A -85,B 0,C 180,E1 -5502.148,E2 -5502.148} C_VEL
LIN {X 0,Y 510.955,Z 256.366,A -85,B 0,C 180,E1 -5502.814,E2 -5502.814} C_VEL
LIN {X 0,Y 511.207,Z 244.634,A -85,B 0,C 180,E1 -5503.364,E2 -5503.364} C_VEL
LIN {X 0,Y 511.5,Z 231.133,A -85,B 0,C 180,E1 -5503.811,E2 -5503.811} C_VEL
LIN {X 0,Y 511.774,Z 217.732,A -85,B 0,C 180,E1 -5504.083,E2 -5504.083} C_VEL
LIN {X 0,Y 511.993,Z 128.102,A -85,B 0,C 180,E1 -5505.355,E2 -5505.355} C_VEL
LIN {X 0,Y 510.187,Z 115.008,A -85,B 0,C 180,E1 -5505.608,E2 -5505.608} C_VEL
LIN {X 0,Y 510.724,Z 93.109,A -85,B 0,C 180,E1 -5508.867,E2 -5508.867} C_VEL
LIN {X 0,Y 511.168,Z 73.779,A -85,B 0,C 180,E1 -5511.791,E2 -5511.791} C_VEL
LIN {X 0,Y 511.643,Z 58.613,A -85,B 0,C 180,E1 -5514.12,E2 -5514.12} C_VEL
LIN {X 0,Y 509.919,Z 48.968,A -85,B 0,C 180,E1 -5515.731,E2 -5515.731} C_VEL
LIN {X 0,Y 509.877,Z 48.974,A -85,B 0,C 180,E1 -5518.844,E2 -5518.844} C_VEL
LIN {X 0,Y 509.82,Z 48.98,A -85,B 0,C 180,E1 -5521.59,E2 -5521.59} C_VEL
LIN {X 0,Y 509.845,Z 48.976,A -85,B 0,C 180,E1 -5524.413,E2 -5524.413} C_VEL
LIN {X 0,Y 509.819,Z 48.978,A -85,B 0,C 180,E1 -5527.34,E2 -5527.34} C_VEL
LIN {X 0,Y 509.837,Z 48.976,A -85,B 0,C 180,E1 -5530.382,E2 -5530.382} C_VEL
LIN {X 0,Y 509.822,Z 48.977,A -85,B 0,C 180,E1 -5533.062,E2 -5533.062} C_VEL
LIN {X 0,Y 509.821,Z 48.977,A -85,B 0,C 180,E1 -5535.793,E2 -5535.793} C_VEL
LIN {X 0,Y 509.864,Z 48.97,A -85,B 0,C 180,E1 -5538.575,E2 -5538.575} C_VEL
LIN {X 0,Y 509.851,Z 48.972,A -85,B 0,C 180,E1 -5541.786,E2 -5541.786} C_VEL
LIN {X 0,Y 509.845,Z 48.974,A -85,B 0,C 180,E1 -5544.623,E2 -5544.623} C_VEL
LIN {X 0,Y 509.861,Z 48.974,A -85,B 0,C 180,E1 -5547.481,E2 -5547.481} C_VEL
LIN {X 0,Y 509.856,Z 48.971,A -85,B 0,C 180,E1 -5550.273,E2 -5550.273} C_VEL
LIN {X 0,Y 509.883,Z 48.972,A -85,B 0,C 180,E1 -5552.944,E2 -5552.944} C_VEL
LIN {X 0,Y 509.868,Z 48.97,A -85,B 0,C 180,E1 -5555.574,E2 -5555.574} C_VEL
LIN {X 0,Y 509.82,Z 48.974,A -85,B 0,C 180,E1 -5558.149,E2 -5558.149} C_VEL
LIN {X 0,Y 509.862,Z 48.975,A -85,B 0,C 180,E1 -5560.682,E2 -5560.682} C_VEL
LIN {X 0,Y 509.882,Z 48.967,A -85,B 0,C 180,E1 -5563.175,E2 -5563.175} C_VEL
LIN {X 0,Y 509.862,Z 48.971,A -85,B 0,C 180,E1 -5565.634,E2 -5565.634} C_VEL
LIN {X 0,Y 509.912,Z 48.965,A -85,B 0,C 180,E1 -5568.875,E2 -5568.875} C_VEL
LIN {X 0,Y 509.949,Z 48.963,A -85,B 0,C 180,E1 -5572.079,E2 -5572.079} C_VEL
LIN {X 0,Y 509.979,Z 48.958,A -85,B 0,C 180,E1 -5574.464,E2 -5574.464} C_VEL
LIN {X 0,Y 510.051,Z 48.95,A -85,B 0,C 180,E1 -5577.631,E2 -5577.631} C_VEL
LIN {X 0,Y 510.061,Z 48.945,A -85,B 0,C 180,E1 -5580.79,E2 -5580.79} C_VEL
LIN {X 0,Y 509.951,Z 48.958,A -85,B 0,C 180,E1 -5583.16,E2 -5583.16} C_VEL
LIN {X 0,Y 509.95,Z 48.959,A -85,B 0,C 180,E1 -5586.33,E2 -5586.33} C_VEL
LIN {X 0,Y 509.887,Z 48.973,A -85,B 0,C 180,E1 -5589.521,E2 -5589.521} C_VEL
LIN {X 0,Y 509.902,Z 48.964,A -85,B 0,C 180,E1 -5591.932,E2 -5591.932} C_VEL
LIN {X 0,Y 509.892,Z 48.973,A -85,B 0,C 180,E1 -5595.242,E2 -5595.242} C_VEL
LIN {X 0,Y 509.865,Z 48.967,A -85,B 0,C 180,E1 -5597.994,E2 -5597.994} C_VEL
LIN {X 0,Y 509.885,Z 48.97,A -85,B 0,C 180,E1 -5600.402,E2 -5600.402} C_VEL
LIN {X 0,Y 509.827,Z 48.975,A -85,B 0,C 180,E1 -5603.564,E2 -5603.564} C_VEL
LIN {X 0,Y 509.877,Z 48.971,A -85,B 0,C 180,E1 -5606.371,E2 -5606.371} C_VEL
LIN {X 0,Y 509.857,Z 48.97,A -85,B 0,C 180,E1 -5609.727,E2 -5609.727} C_VEL
LIN {X 0,Y 509.866,Z 48.973,A -85,B 0,C 180,E1 -5612.773,E2 -5612.773} C_VEL
LIN {X 0,Y 509.821,Z 48.975,A -85,B 0,C 180,E1 -5615.578,E2 -5615.578} C_VEL
LIN {X 0,Y 509.848,Z 48.979,A -85,B 0,C 180,E1 -5618.339,E2 -5618.339} C_VEL
LIN {X 0,Y 509.831,Z 48.973,A -85,B 0,C 180,E1 -5621.429,E2 -5621.429} C_VEL
LIN {X 0,Y 509.839,Z 48.973,A -85,B 0,C 180,E1 -5624.671,E2 -5624.671} C_VEL
LIN {X 0,Y 509.803,Z 48.986,A -85,B 0,C 180,E1 -5627.508,E2 -5627.508} C_VEL
LIN {X 0,Y 509.832,Z 48.976,A -85,B 0,C 180,E1 -5630.647,E2 -5630.647} C_VEL
LIN {X 0,Y 509.802,Z 48.985,A -85,B 0,C 180,E1 -5633.73,E2 -5633.73} C_VEL
LIN {X 0,Y 509.122,Z 49.067,A -85,B 0,C 180,E1 -5634.17,E2 -5634.17} C_VEL
LIN {X 0,Y 506.284,Z 49.421,A -85,B 0,C 180,E1 -5634.859,E2 -5634.859} C_VEL
LIN {X 0,Y 503.45,Z 49.777,A -85,B 0,C 180,E1 -5635.555,E2 -5635.555} C_VEL
LIN {X 0,Y 502.792,Z 49.859,A -85,B 0,C 180,E1 -5636.004,E2 -5636.004} C_VEL
LIN {X 0,Y 502.847,Z 49.909,A -85,B 0,C 180,E1 -5637.148,E2 -5637.148} C_VEL
LIN {X 0,Y 503.627,Z 55.371,A -85,B 0,C 180,E1 -5638.348,E2 -5638.348} C_VEL
LIN {X 0,Y 503.435,Z 64.635,A -85,B 0,C 180,E1 -5640.249,E2 -5640.249} C_VEL
LIN {X 0,Y 505.577,Z 74.687,A -85,B 0,C 180,E1 -5640.47,E2 -5640.47} C_VEL
LIN {X 0,Y 504.956,Z 170.861,A -85,B 0,C 180,E1 -5641.87,E2 -5641.87} C_VEL
LIN {X 0,Y 504.793,Z 184.04,A -85,B 0,C 180,E1 -5642.227,E2 -5642.227} C_VEL
LIN {X 0,Y 504.578,Z 196.131,A -85,B 0,C 180,E1 -5642.711,E2 -5642.711} C_VEL
LIN {X 0,Y 504.279,Z 206.773,A -85,B 0,C 180,E1 -5643.276,E2 -5643.276} C_VEL
LIN {X 0,Y 503.87,Z 218.14,A -85,B 0,C 180,E1 -5644.048,E2 -5644.048} C_VEL
LIN {X 0,Y 503.59,Z 228.286,A -85,B 0,C 180,E1 -5644.917,E2 -5644.917} C_VEL
LIN {X 0,Y 503.269,Z 237.593,A -85,B 0,C 180,E1 -5645.892,E2 -5645.892} C_VEL
LIN {X 0,Y 502.958,Z 246.005,A -85,B 0,C 180,E1 -5646.968,E2 -5646.968} C_VEL
LIN {X 0,Y 502.715,Z 252.871,A -85,B 0,C 180,E1 -5648.04,E2 -5648.04} C_VEL
LIN {X 0,Y 502.523,Z 258.486,A -85,B 0,C 180,E1 -5649.107,E2 -5649.107} C_VEL
LIN {X 0,Y 502.38,Z 263.888,A -85,B 0,C 180,E1 -5650.382,E2 -5650.382} C_VEL
LIN {X 0,Y 502.253,Z 267.99,A -85,B 0,C 180,E1 -5651.649,E2 -5651.649} C_VEL
LIN {X 0,Y 502.133,Z 270.956,A -85,B 0,C 180,E1 -5652.907,E2 -5652.907} C_VEL
LIN {X 0,Y 502.094,Z 272.333,A -85,B 0,C 180,E1 -5653.743,E2 -5653.743} C_VEL
LIN {X 0,Y 502.101,Z 273.594,A -85,B 0,C 180,E1 -5654.975,E2 -5654.975} C_VEL
LIN {X 0,Y 502.066,Z 273.926,A -85,B 0,C 180,E1 -5656.234,E2 -5656.234} C_VEL
LIN {X 0,Y 502.098,Z 273.612,A -85,B 0,C 180,E1 -5657.059,E2 -5657.059} C_VEL
LIN {X 0,Y 502.165,Z 272.178,A -85,B 0,C 180,E1 -5658.432,E2 -5658.432} C_VEL
LIN {X 0,Y 502.216,Z 270.196,A -85,B 0,C 180,E1 -5659.519,E2 -5659.519} C_VEL
LIN {X 0,Y 502.272,Z 267.042,A -85,B 0,C 180,E1 -5660.74,E2 -5660.74} C_VEL
LIN {X 0,Y 502.398,Z 262.823,A -85,B 0,C 180,E1 -5661.959,E2 -5661.959} C_VEL
LIN {X 0,Y 502.536,Z 257.346,A -85,B 0,C 180,E1 -5663.192,E2 -5663.192} C_VEL
LIN {X 0,Y 502.775,Z 250.709,A -85,B 0,C 180,E1 -5664.385,E2 -5664.385} C_VEL
LIN {X 0,Y 503.032,Z 242.369,A -85,B 0,C 180,E1 -5665.593,E2 -5665.593} C_VEL
LIN {X 0,Y 503.325,Z 233.794,A -85,B 0,C 180,E1 -5666.598,E2 -5666.598} C_VEL
LIN {X 0,Y 503.692,Z 223.257,A -85,B 0,C 180,E1 -5667.601,E2 -5667.601} C_VEL
LIN {X 0,Y 504.077,Z 212.783,A -85,B 0,C 180,E1 -5668.402,E2 -5668.402} C_VEL
LIN {X 0,Y 504.396,Z 201.173,A -85,B 0,C 180,E1 -5669.102,E2 -5669.102} C_VEL
LIN {X 0,Y 504.644,Z 187.904,A -85,B 0,C 180,E1 -5669.701,E2 -5669.701} C_VEL
LIN {X 0,Y 504.864,Z 175.078,A -85,B 0,C 180,E1 -5670.1,E2 -5670.1} C_VEL
LIN {X 0,Y 505.024,Z 159.665,A -85,B 0,C 180,E1 -5670.374,E2 -5670.374} C_VEL
LIN {X 0,Y 505.322,Z 73.907,A -85,B 0,C 180,E1 -5671.606,E2 -5671.606} C_VEL
LIN {X 0,Y 503.318,Z 64.104,A -85,B 0,C 180,E1 -5671.826,E2 -5671.826} C_VEL
LIN {X 0,Y 503.463,Z 53.653,A -85,B 0,C 180,E1 -5674.003,E2 -5674.003} C_VEL
LIN {X 0,Y 502.872,Z 49.849,A -85,B 0,C 180,E1 -5674.861,E2 -5674.861} C_VEL
LIN {X 0,Y 502.94,Z 49.836,A -85,B 0,C 180,E1 -5677.225,E2 -5677.225} C_VEL
LIN {X 0,Y 502.82,Z 49.854,A -85,B 0,C 180,E1 -5680.469,E2 -5680.469} C_VEL
LIN {X 0,Y 502.835,Z 49.848,A -85,B 0,C 180,E1 -5682.922,E2 -5682.922} C_VEL
LIN {X 0,Y 502.855,Z 49.842,A -85,B 0,C 180,E1 -5685.4,E2 -5685.4} C_VEL
LIN {X 0,Y 502.832,Z 49.848,A -85,B 0,C 180,E1 -5688.752,E2 -5688.752} C_VEL
LIN {X 0,Y 502.789,Z 49.851,A -85,B 0,C 180,E1 -5691.311,E2 -5691.311} C_VEL
LIN {X 0,Y 502.782,Z 49.857,A -85,B 0,C 180,E1 -5693.914,E2 -5693.914} C_VEL
LIN {X 0,Y 502.87,Z 49.842,A -85,B 0,C 180,E1 -5696.566,E2 -5696.566} C_VEL
LIN {X 0,Y 502.828,Z 49.847,A -85,B 0,C 180,E1 -5699.288,E2 -5699.288} C_VEL
LIN {X 0,Y 502.789,Z 49.856,A -85,B 0,C 180,E1 -5702.084,E2 -5702.084} C_VEL
LIN {X 0,Y 502.813,Z 49.848,A -85,B 0,C 180,E1 -5704.965,E2 -5704.965} C_VEL
LIN {X 0,Y 502.798,Z 49.854,A -85,B 0,C 180,E1 -5707.954,E2 -5707.954} C_VEL
LIN {X 0,Y 502.824,Z 49.849,A -85,B 0,C 180,E1 -5711.066,E2 -5711.066} C_VEL
LIN {X 0,Y 502.79,Z 49.851,A -85,B 0,C 180,E1 -5714.53,E2 -5714.53} C_VEL
LIN {X 0,Y 502.799,Z 49.851,A -85,B 0,C 180,E1 -5717.86,E2 -5717.86} C_VEL
LIN {X 0,Y 502.806,Z 49.855,A -85,B 0,C 180,E1 -5721.024,E2 -5721.024} C_VEL
LIN {X 0,Y 502.779,Z 49.852,A -85,B 0,C 180,E1 -5724.169,E2 -5724.169} C_VEL
LIN {X 0,Y 502.836,Z 49.853,A -85,B 0,C 180,E1 -5726.993,E2 -5726.993} C_VEL
LIN {X 0,Y 502.818,Z 49.847,A -85,B 0,C 180,E1 -5730.065,E2 -5730.065} C_VEL
LIN {X 0,Y 502.836,Z 49.85,A -85,B 0,C 180,E1 -5732.533,E2 -5732.533} C_VEL
LIN {X 0,Y 502.832,Z 49.846,A -85,B 0,C 180,E1 -5735.298,E2 -5735.298} C_VEL
LIN {X 0,Y 502.784,Z 49.852,A -85,B 0,C 180,E1 -5737.826,E2 -5737.826} C_VEL
LIN {X 0,Y 502.828,Z 49.853,A -85,B 0,C 180,E1 -5740.4,E2 -5740.4} C_VEL
LIN {X 0,Y 502.833,Z 49.847,A -85,B 0,C 180,E1 -5742.931,E2 -5742.931} C_VEL
LIN {X 0,Y 502.848,Z 49.843,A -85,B 0,C 180,E1 -5745.429,E2 -5745.429} C_VEL
LIN {X 0,Y 502.88,Z 49.841,A -85,B 0,C 180,E1 -5748.717,E2 -5748.717} C_VEL
LIN {X 0,Y 502.903,Z 49.844,A -85,B 0,C 180,E1 -5751.966,E2 -5751.966} C_VEL
LIN {X 0,Y 502.937,Z 49.835,A -85,B 0,C 180,E1 -5754.386,E2 -5754.386} C_VEL
LIN {X 0,Y 503.025,Z 49.826,A -85,B 0,C 180,E1 -5757.598,E2 -5757.598} C_VEL
LIN {X 0,Y 503.029,Z 49.826,A -85,B 0,C 180,E1 -5760,E2 -5760} C_VEL
LIN {X 0,Y 503.024,Z 49.822,A -85,B 0,C 180,E1 -5762.402,E2 -5762.402} C_VEL
LIN {X 0,Y 502.933,Z 49.841,A -85,B 0,C 180,E1 -5765.613,E2 -5765.613} C_VEL
LIN {X 0,Y 502.883,Z 49.841,A -85,B 0,C 180,E1 -5768.033,E2 -5768.033} C_VEL
LIN {X 0,Y 502.879,Z 49.847,A -85,B 0,C 180,E1 -5771.283,E2 -5771.283} C_VEL
LIN {X 0,Y 502.846,Z 49.844,A -85,B 0,C 180,E1 -5774.571,E2 -5774.571} C_VEL
LIN {X 0,Y 502.824,Z 49.847,A -85,B 0,C 180,E1 -5777.908,E2 -5777.908} C_VEL
LIN {X 0,Y 502.831,Z 49.847,A -85,B 0,C 180,E1 -5780.536,E2 -5780.536} C_VEL
LIN {X 0,Y 502.792,Z 49.858,A -85,B 0,C 180,E1 -5783.04,E2 -5783.04} C_VEL
LIN {X 0,Y 502.813,Z 49.848,A -85,B 0,C 180,E1 -5785.677,E2 -5785.677} C_VEL
LIN {X 0,Y 502.837,Z 49.848,A -85,B 0,C 180,E1 -5788.373,E2 -5788.373} C_VEL
LIN {X 0,Y 502.794,Z 49.85,A -85,B 0,C 180,E1 -5791.499,E2 -5791.499} C_VEL
LIN {X 0,Y 502.805,Z 49.85,A -85,B 0,C 180,E1 -5793.994,E2 -5793.994} C_VEL
LIN {X 0,Y 502.779,Z 49.853,A -85,B 0,C 180,E1 -5797.178,E2 -5797.178} C_VEL
LIN {X 0,Y 502.789,Z 49.854,A -85,B 0,C 180,E1 -5800.015,E2 -5800.015} C_VEL
LIN {X 0,Y 502.805,Z 49.856,A -85,B 0,C 180,E1 -5802.199,E2 -5802.199} C_VEL
LIN {X 0,Y 502.787,Z 49.852,A -85,B 0,C 180,E1 -5805.47,E2 -5805.47} C_VEL
LIN {X 0,Y 502.822,Z 49.847,A -85,B 0,C 180,E1 -5808.934,E2 -5808.934} C_VEL
LIN {X 0,Y 502.795,Z 49.857,A -85,B 0,C 180,E1 -5812.046,E2 -5812.046} C_VEL
LIN {X 0,Y 502.801,Z 49.849,A -85,B 0,C 180,E1 -5815.034,E2 -5815.034} C_VEL
LIN {X 0,Y 502.785,Z 49.857,A -85,B 0,C 180,E1 -5817.915,E2 -5817.915} C_VEL
LIN {X 0,Y 502.826,Z 49.851,A -85,B 0,C 180,E1 -5820.712,E2 -5820.712} C_VEL
LIN {X 0,Y 502.881,Z 49.847,A -85,B 0,C 180,E1 -5824.104,E2 -5824.104} C_VEL
LIN {X 0,Y 502.913,Z 49.985,A -85,B 0,C 180,E1 -5824.217,E2 -5824.217} C_VEL
LIN {X 0,Y 504.581,Z 59.235,A -85,B 0,C 180,E1 -5825.739,E2 -5825.739} C_VEL
LIN {X 0,Y 504.159,Z 76.002,A -85,B 0,C 180,E1 -5828.32,E2 -5828.32} C_VEL
LIN {X 0,Y 503.583,Z 97.764,A -85,B 0,C 180,E1 -5831.624,E2 -5831.624} C_VEL
LIN {X 0,Y 503.163,Z 115,A -85,B 0,C 180,E1 -5834.199,E2 -5834.199} C_VEL
LIN {X 0,Y 505.288,Z 130.744,A -85,B 0,C 180,E1 -5834.49,E2 -5834.49} C_VEL
LIN {X 0,Y 504.798,Z 224.209,A -85,B 0,C 180,E1 -5835.847,E2 -5835.847} C_VEL
LIN {X 0,Y 504.484,Z 237.325,A -85,B 0,C 180,E1 -5836.198,E2 -5836.198} C_VEL
LIN {X 0,Y 504.147,Z 249.995,A -85,B 0,C 180,E1 -5836.702,E2 -5836.702} C_VEL
LIN {X 0,Y 503.82,Z 261.324,A -85,B 0,C 180,E1 -5837.312,E2 -5837.312} C_VEL
LIN {X 0,Y 503.389,Z 272.938,A -85,B 0,C 180,E1 -5838.116,E2 -5838.116} C_VEL
LIN {X 0,Y 503.082,Z 283.448,A -85,B 0,C 180,E1 -5839.027,E2 -5839.027} C_VEL
LIN {X 0,Y 502.779,Z 292.041,A -85,B 0,C 180,E1 -5839.937,E2 -5839.937} C_VEL
LIN {X 0,Y 502.528,Z 299.972,A -85,B 0,C 180,E1 -5840.948,E2 -5840.948} C_VEL
LIN {X 0,Y 502.355,Z 307.724,A -85,B 0,C 180,E1 -5842.16,E2 -5842.16} C_VEL
LIN {X 0,Y 502.187,Z 314.863,A -85,B 0,C 180,E1 -5843.572,E2 -5843.572} C_VEL
LIN {X 0,Y 502.168,Z 319.619,A -85,B 0,C 180,E1 -5844.78,E2 -5844.78} C_VEL
LIN {X 0,Y 502.164,Z 323.251,A -85,B 0,C 180,E1 -5845.987,E2 -5845.987} C_VEL
LIN {X 0,Y 502.158,Z 325.124,A -85,B 0,C 180,E1 -5846.79,E2 -5846.79} C_VEL
LIN {X 0,Y 502.128,Z 326.526,A -85,B 0,C 180,E1 -5847.593,E2 -5847.593} C_VEL
LIN {X 0,Y 502.016,Z 328.129,A -85,B 0,C 180,E1 -5849.198,E2 -5849.198} C_VEL
LIN {X 0,Y 502.017,Z 328.344,A -85,B 0,C 180,E1 -5850,E2 -5850} C_VEL
LIN {X 0,Y 502.043,Z 327.508,A -85,B 0,C 180,E1 -5851.604,E2 -5851.604} C_VEL
LIN {X 0,Y 502.128,Z 326.507,A -85,B 0,C 180,E1 -5852.406,E2 -5852.406} C_VEL
LIN {X 0,Y 502.158,Z 325.098,A -85,B 0,C 180,E1 -5853.209,E2 -5853.209} C_VEL
LIN {X 0,Y 502.102,Z 322.132,A -85,B 0,C 180,E1 -5854.415,E2 -5854.415} C_VEL
LIN {X 0,Y 502.183,Z 318.128,A -85,B 0,C 180,E1 -5855.622,E2 -5855.622} C_VEL
LIN {X 0,Y 502.271,Z 312.072,A -85,B 0,C 180,E1 -5857.012,E2 -5857.012} C_VEL
LIN {X 0,Y 502.413,Z 305.247,A -85,B 0,C 180,E1 -5858.243,E2 -5858.243} C_VEL
LIN {X 0,Y 502.633,Z 296.911,A -85,B 0,C 180,E1 -5859.456,E2 -5859.456} C_VEL
LIN {X 0,Y 502.923,Z 288.374,A -85,B 0,C 180,E1 -5860.466,E2 -5860.466} C_VEL
LIN {X 0,Y 503.301,Z 277.843,A -85,B 0,C 180,E1 -5861.477,E2 -5861.477} C_VEL
LIN {X 0,Y 503.613,Z 266.568,A -85,B 0,C 180,E1 -5862.349,E2 -5862.349} C_VEL
LIN {X 0,Y 504.019,Z 254.104,A -85,B 0,C 180,E1 -5863.096,E2 -5863.096} C_VEL
LIN {X 0,Y 504.365,Z 241.746,A -85,B 0,C 180,E1 -5863.651,E2 -5863.651} C_VEL
LIN {X 0,Y 504.681,Z 229.086,A -85,B 0,C 180,E1 -5864.053,E2 -5864.053} C_VEL
LIN {X 0,Y 504.884,Z 215.925,A -85,B 0,C 180,E1 -5864.304,E2 -5864.304} C_VEL
LIN {X 0,Y 505.195,Z 129.004,A -85,B 0,C 180,E1 -5865.555,E2 -5865.555} C_VEL
LIN {X 0,Y 503.174,Z 114.64,A -85,B 0,C 180,E1 -5865.836,E2 -5865.836} C_VEL
LIN {X 0,Y 503.741,Z 94.192,A -85,B 0,C 180,E1 -5868.927,E2 -5868.927} C_VEL
LIN {X 0,Y 504.269,Z 73.525,A -85,B 0,C 180,E1 -5872.104,E2 -5872.104} C_VEL
LIN {X 0,Y 504.728,Z 59.763,A -85,B 0,C 180,E1 -5874.253,E2 -5874.253} C_VEL
LIN {X 0,Y 502.893,Z 49.845,A -85,B 0,C 180,E1 -5875.95,E2 -5875.95} C_VEL
LIN {X 0,Y 502.825,Z 49.851,A -85,B 0,C 180,E1 -5879.287,E2 -5879.287} C_VEL
LIN {X 0,Y 502.782,Z 49.861,A -85,B 0,C 180,E1 -5882.084,E2 -5882.084} C_VEL
LIN {X 0,Y 502.806,Z 49.849,A -85,B 0,C 180,E1 -5884.965,E2 -5884.965} C_VEL
LIN {X 0,Y 502.793,Z 49.859,A -85,B 0,C 180,E1 -5887.953,E2 -5887.953} C_VEL
LIN {X 0,Y 502.818,Z 49.849,A -85,B 0,C 180,E1 -5891.066,E2 -5891.066} C_VEL
LIN {X 0,Y 502.784,Z 49.85,A -85,B 0,C 180,E1 -5894.53,E2 -5894.53} C_VEL
LIN {X 0,Y 502.798,Z 49.854,A -85,B 0,C 180,E1 -5897.861,E2 -5897.861} C_VEL
LIN {X 0,Y 502.819,Z 49.848,A -85,B 0,C 180,E1 -5900.241,E2 -5900.241} C_VEL
LIN {X 0,Y 502.776,Z 49.856,A -85,B 0,C 180,E1 -5903.053,E2 -5903.053} C_VEL
LIN {X 0,Y 502.806,Z 49.848,A -85,B 0,C 180,E1 -5906.006,E2 -5906.006} C_VEL
LIN {X 0,Y 502.794,Z 49.856,A -85,B 0,C 180,E1 -5908.857,E2 -5908.857} C_VEL
LIN {X 0,Y 502.842,Z 49.845,A -85,B 0,C 180,E1 -5911.705,E2 -5911.705} C_VEL
LIN {X 0,Y 502.838,Z 49.845,A -85,B 0,C 180,E1 -5914.324,E2 -5914.324} C_VEL
LIN {X 0,Y 502.808,Z 49.846,A -85,B 0,C 180,E1 -5917.295,E2 -5917.295} C_VEL
LIN {X 0,Y 502.823,Z 49.853,A -85,B 0,C 180,E1 -5920.4,E2 -5920.4} C_VEL
LIN {X 0,Y 502.832,Z 49.847,A -85,B 0,C 180,E1 -5922.932,E2 -5922.932} C_VEL
LIN {X 0,Y 502.843,Z 49.844,A -85,B 0,C 180,E1 -5925.429,E2 -5925.429} C_VEL
LIN {X 0,Y 502.875,Z 49.843,A -85,B 0,C 180,E1 -5928.717,E2 -5928.717} C_VEL
LIN {X 0,Y 502.9,Z 49.841,A -85,B 0,C 180,E1 -5931.967,E2 -5931.967} C_VEL
LIN {X 0,Y 502.933,Z 49.837,A -85,B 0,C 180,E1 -5934.387,E2 -5934.387} C_VEL
LIN {X 0,Y 503.021,Z 49.825,A -85,B 0,C 180,E1 -5937.598,E2 -5937.598} C_VEL
LIN {X 0,Y 503.024,Z 49.827,A -85,B 0,C 180,E1 -5940,E2 -5940} C_VEL
LIN {X 0,Y 503.02,Z 49.819,A -85,B 0,C 180,E1 -5942.402,E2 -5942.402} C_VEL
LIN {X 0,Y 502.929,Z 49.84,A -85,B 0,C 180,E1 -5945.614,E2 -5945.614} C_VEL
LIN {X 0,Y 502.878,Z 49.838,A -85,B 0,C 180,E1 -5948.034,E2 -5948.034} C_VEL
LIN {X 0,Y 502.875,Z 49.847,A -85,B 0,C 180,E1 -5951.283,E2 -5951.283} C_VEL
LIN {X 0,Y 502.842,Z 49.845,A -85,B 0,C 180,E1 -5954.571,E2 -5954.571} C_VEL
LIN {X 0,Y 502.821,Z 49.845,A -85,B 0,C 180,E1 -5957.909,E2 -5957.909} C_VEL
LIN {X 0,Y 502.827,Z 49.851,A -85,B 0,C 180,E1 -5960.537,E2 -5960.537} C_VEL
LIN {X 0,Y 502.789,Z 49.856,A -85,B 0,C 180,E1 -5963.041,E2 -5963.041} C_VEL
LIN {X 0,Y 502.797,Z 49.848,A -85,B 0,C 180,E1 -5965.678,E2 -5965.678} C_VEL
LIN {X 0,Y 502.795,Z 49.857,A -85,B 0,C 180,E1 -5968.376,E2 -5968.376} C_VEL
LIN {X 0,Y 502.795,Z 49.852,A -85,B 0,C 180,E1 -5971.144,E2 -5971.144} C_VEL
LIN {X 0,Y 502.788,Z 49.856,A -85,B 0,C 180,E1 -5973.996,E2 -5973.996} C_VEL
LIN {X 0,Y 502.764,Z 49.855,A -85,B 0,C 180,E1 -5977.176,E2 -5977.176} C_VEL
LIN {X 0,Y 502.77,Z 49.86,A -85,B 0,C 180,E1 -5980.017,E2 -5980.017} C_VEL
LIN {X 0,Y 502.771,Z 49.862,A -85,B 0,C 180,E1 -5982.196,E2 -5982.196} C_VEL
LIN {X 0,Y 502.786,Z 49.855,A -85,B 0,C 180,E1 -5985.471,E2 -5985.471} C_VEL
LIN {X 0,Y 502.795,Z 49.859,A -85,B 0,C 180,E1 -5987.861,E2 -5987.861} C_VEL
LIN {X 0,Y 502.784,Z 49.855,A -85,B 0,C 180,E1 -5991.023,E2 -5991.023} C_VEL
LIN {X 0,Y 502.77,Z 49.858,A -85,B 0,C 180,E1 -5994.171,E2 -5994.171} C_VEL
LIN {X 0,Y 502.792,Z 49.859,A -85,B 0,C 180,E1 -5996.004,E2 -5996.004} C_VEL
LIN {X 0,Y 502.529,Z 50.169,A -85,B 0,C 180,E1 -5996.448,E2 -5996.448} C_VEL
LIN {X 0,Y 501.372,Z 51.571,A -85,B 0,C 180,E1 -5997.089,E2 -5997.089} C_VEL
LIN {X 0,Y 499.758,Z 53.76,A -85,B 0,C 180,E1 -5997.696,E2 -5997.696} C_VEL
LIN {X 0,Y 497.614,Z 57.476,A -85,B 0,C 180,E1 -5998.493,E2 -5998.493} C_VEL
LIN {X 0,Y 496.555,Z 61.452,A -85,B 0,C 180,E1 -5999.298,E2 -5999.298} C_VEL
LIN {X 0,Y 496.495,Z 64.729,A -85,B 0,C 180,E1 -5999.991,E2 -5999.991} C_VEL
LIN {X 0,Y 498.775,Z 76.228,A -85,B 0,C 180,E1 -6000.256,E2 -6000.256} C_VEL
LIN {X 0,Y 498.136,Z 170.836,A -85,B 0,C 180,E1 -6001.651,E2 -6001.651} C_VEL
LIN {X 0,Y 497.958,Z 184.145,A -85,B 0,C 180,E1 -6002.013,E2 -6002.013} C_VEL
LIN {X 0,Y 497.706,Z 196.59,A -85,B 0,C 180,E1 -6002.516,E2 -6002.516} C_VEL
LIN {X 0,Y 497.378,Z 207.697,A -85,B 0,C 180,E1 -6003.118,E2 -6003.118} C_VEL
LIN {X 0,Y 496.943,Z 218.731,A -85,B 0,C 180,E1 -6003.885,E2 -6003.885} C_VEL
LIN {X 0,Y 496.632,Z 228.857,A -85,B 0,C 180,E1 -6004.767,E2 -6004.767} C_VEL
LIN {X 0,Y 496.287,Z 238.107,A -85,B 0,C 180,E1 -6005.753,E2 -6005.753} C_VEL
LIN {X 0,Y 495.956,Z 246.998,A -85,B 0,C 180,E1 -6006.918,E2 -6006.918} C_VEL
LIN {X 0,Y 495.625,Z 254.522,A -85,B 0,C 180,E1 -6008.147,E2 -6008.147} C_VEL
LIN {X 0,Y 495.445,Z 260.785,A -85,B 0,C 180,E1 -6009.429,E2 -6009.429} C_VEL
LIN {X 0,Y 495.268,Z 266.513,A -85,B 0,C 180,E1 -6010.951,E2 -6010.951} C_VEL
LIN {X 0,Y 495.15,Z 269.424,A -85,B 0,C 180,E1 -6011.987,E2 -6011.987} C_VEL
LIN {X 0,Y 495.022,Z 272.447,A -85,B 0,C 180,E1 -6013.504,E2 -6013.504} C_VEL
LIN {X 0,Y 495.01,Z 273.945,A -85,B 0,C 180,E1 -6014.896,E2 -6014.896} C_VEL
LIN {X 0,Y 494.999,Z 274.342,A -85,B 0,C 180,E1 -6016.033,E2 -6016.033} C_VEL
LIN {X 0,Y 495.003,Z 274.113,A -85,B 0,C 180,E1 -6016.87,E2 -6016.87} C_VEL
LIN {X 0,Y 495.085,Z 272.672,A -85,B 0,C 180,E1 -6018.379,E2 -6018.379} C_VEL
LIN {X 0,Y 495.132,Z 271.003,A -85,B 0,C 180,E1 -6019.367,E2 -6019.367} C_VEL
LIN {X 0,Y 495.179,Z 268.011,A -85,B 0,C 180,E1 -6020.607,E2 -6020.607} C_VEL
LIN {X 0,Y 495.316,Z 263.963,A -85,B 0,C 180,E1 -6021.843,E2 -6021.843} C_VEL
LIN {X 0,Y 495.489,Z 258.333,A -85,B 0,C 180,E1 -6023.163,E2 -6023.163} C_VEL
LIN {X 0,Y 495.735,Z 251.015,A -85,B 0,C 180,E1 -6024.509,E2 -6024.509} C_VEL
LIN {X 0,Y 496.026,Z 242.643,A -85,B 0,C 180,E1 -6025.734,E2 -6025.734} C_VEL
LIN {X 0,Y 496.36,Z 234.034,A -85,B 0,C 180,E1 -6026.754,E2 -6026.754} C_VEL
LIN {X 0,Y 496.745,Z 223.463,A -85,B 0,C 180,E1 -6027.771,E2 -6027.771} C_VEL
LIN {X 0,Y 497.138,Z 212.949,A -85,B 0,C 180,E1 -6028.583,E2 -6028.583} C_VEL
LIN {X 0,Y 497.475,Z 201.25,A -85,B 0,C 180,E1 -6029.292,E2 -6029.292} C_VEL
LIN {X 0,Y 497.74,Z 189.138,A -85,B 0,C 180,E1 -6029.849,E2 -6029.849} C_VEL
LIN {X 0,Y 497.956,Z 176.757,A -85,B 0,C 180,E1 -6030.253,E2 -6030.253} C_VEL
LIN {X 0,Y 498.107,Z 164.16,A -85,B 0,C 180,E1 -6030.506,E2 -6030.506} C_VEL
LIN {X 0,Y 498.512,Z 75.019,A -85,B 0,C 180,E1 -6031.801,E2 -6031.801} C_VEL
LIN {X 0,Y 496.324,Z 64.503,A -85,B 0,C 180,E1 -6032.029,E2 -6032.029} C_VEL
LIN {X 0,Y 496.469,Z 54.831,A -85,B 0,C 180,E1 -6034.059,E2 -6034.059} C_VEL
LIN {X 0,Y 495.847,Z 50.724,A -85,B 0,C 180,E1 -6034.981,E2 -6034.981} C_VEL
LIN {X 0,Y 495.912,Z 50.711,A -85,B 0,C 180,E1 -6037.328,E2 -6037.328} C_VEL
LIN {X 0,Y 495.797,Z 50.722,A -85,B 0,C 180,E1 -6039.794,E2 -6039.794} C_VEL
LIN {X 0,Y 495.795,Z 50.727,A -85,B 0,C 180,E1 -6042.277,E2 -6042.277} C_VEL
LIN {X 0,Y 495.83,Z 50.718,A -85,B 0,C 180,E1 -6045.452,E2 -6045.452} C_VEL
LIN {X 0,Y 495.785,Z 50.731,A -85,B 0,C 180,E1 -6048.237,E2 -6048.237} C_VEL
LIN {X 0,Y 495.78,Z 50.726,A -85,B 0,C 180,E1 -6050.756,E2 -6050.756} C_VEL
LIN {X 0,Y 495.749,Z 50.728,A -85,B 0,C 180,E1 -6053.387,E2 -6053.387} C_VEL
LIN {X 0,Y 495.829,Z 50.718,A -85,B 0,C 180,E1 -6056.749,E2 -6056.749} C_VEL
LIN {X 0,Y 495.771,Z 50.731,A -85,B 0,C 180,E1 -6059.746,E2 -6059.746} C_VEL
LIN {X 0,Y 495.773,Z 50.725,A -85,B 0,C 180,E1 -6062.594,E2 -6062.594} C_VEL
LIN {X 0,Y 495.761,Z 50.732,A -85,B 0,C 180,E1 -6065.537,E2 -6065.537} C_VEL
LIN {X 0,Y 495.767,Z 50.726,A -85,B 0,C 180,E1 -6068.768,E2 -6068.768} C_VEL
LIN {X 0,Y 495.76,Z 50.731,A -85,B 0,C 180,E1 -6071.781,E2 -6071.781} C_VEL
LIN {X 0,Y 495.741,Z 50.734,A -85,B 0,C 180,E1 -6075.141,E2 -6075.141} C_VEL
LIN {X 0,Y 495.76,Z 50.726,A -85,B 0,C 180,E1 -6078.219,E2 -6078.219} C_VEL
LIN {X 0,Y 495.755,Z 50.732,A -85,B 0,C 180,E1 -6081.408,E2 -6081.408} C_VEL
LIN {X 0,Y 495.752,Z 50.729,A -85,B 0,C 180,E1 -6084.462,E2 -6084.462} C_VEL
LIN {X 0,Y 495.771,Z 50.727,A -85,B 0,C 180,E1 -6087.405,E2 -6087.405} C_VEL
LIN {X 0,Y 495.77,Z 50.727,A -85,B 0,C 180,E1 -6090.253,E2 -6090.253} C_VEL
LIN {X 0,Y 495.827,Z 50.72,A -85,B 0,C 180,E1 -6093.251,E2 -6093.251} C_VEL
LIN {X 0,Y 495.756,Z 50.727,A -85,B 0,C 180,E1 -6095.725,E2 -6095.725} C_VEL
LIN {X 0,Y 495.746,Z 50.734,A -85,B 0,C 180,E1 -6098.371,E2 -6098.371} C_VEL
LIN {X 0,Y 495.787,Z 50.725,A -85,B 0,C 180,E1 -6100.971,E2 -6100.971} C_VEL
LIN {X 0,Y 495.781,Z 50.724,A -85,B 0,C 180,E1 -6103.53,E2 -6103.53} C_VEL
LIN {X 0,Y 495.796,Z 50.727,A -85,B 0,C 180,E1 -6106.055,E2 -6106.055} C_VEL
LIN {X 0,Y 495.855,Z 50.718,A -85,B 0,C 180,E1 -6108.555,E2 -6108.555} C_VEL
LIN {X 0,Y 495.875,Z 50.717,A -85,B 0,C 180,E1 -6111.852,E2 -6111.852} C_VEL
LIN {X 0,Y 495.893,Z 50.714,A -85,B 0,C 180,E1 -6114.306,E2 -6114.306} C_VEL
LIN {X 0,Y 495.994,Z 50.701,A -85,B 0,C 180,E1 -6117.564,E2 -6117.564} C_VEL
LIN {X 0,Y 495.985,Z 50.698,A -85,B 0,C 180,E1 -6120.812,E2 -6120.812} C_VEL
LIN {X 0,Y 495.993,Z 50.698,A -85,B 0,C 180,E1 -6122.436,E2 -6122.436} C_VEL
LIN {X 0,Y 495.889,Z 50.717,A -85,B 0,C 180,E1 -6125.693,E2 -6125.693} C_VEL
LIN {X 0,Y 495.839,Z 50.718,A -85,B 0,C 180,E1 -6128.148,E2 -6128.148} C_VEL
LIN {X 0,Y 495.853,Z 50.722,A -85,B 0,C 180,E1 -6131.445,E2 -6131.445} C_VEL
LIN {X 0,Y 495.792,Z 50.725,A -85,B 0,C 180,E1 -6134.783,E2 -6134.783} C_VEL
LIN {X 0,Y 495.767,Z 50.732,A -85,B 0,C 180,E1 -6137.319,E2 -6137.319} C_VEL
LIN {X 0,Y 495.773,Z 50.725,A -85,B 0,C 180,E1 -6139.89,E2 -6139.89} C_VEL
LIN {X 0,Y 495.762,Z 50.733,A -85,B 0,C 180,E1 -6142.861,E2 -6142.861} C_VEL
LIN {X 0,Y 495.768,Z 50.726,A -85,B 0,C 180,E1 -6146.069,E2 -6146.069} C_VEL
LIN {X 0,Y 495.771,Z 50.733,A -85,B 0,C 180,E1 -6148.815,E2 -6148.815} C_VEL
LIN {X 0,Y 495.757,Z 50.727,A -85,B 0,C 180,E1 -6151.725,E2 -6151.725} C_VEL
LIN {X 0,Y 495.771,Z 50.732,A -85,B 0,C 180,E1 -6154.694,E2 -6154.694} C_VEL
LIN {X 0,Y 495.731,Z 50.73,A -85,B 0,C 180,E1 -6157.562,E2 -6157.562} C_VEL
LIN {X 0,Y 495.768,Z 50.729,A -85,B 0,C 180,E1 -6160.7,E2 -6160.7} C_VEL
LIN {X 0,Y 495.73,Z 50.735,A -85,B 0,C 180,E1 -6164.002,E2 -6164.002} C_VEL
LIN {X 0,Y 495.727,Z 50.73,A -85,B 0,C 180,E1 -6167.117,E2 -6167.117} C_VEL
LIN {X 0,Y 495.76,Z 50.734,A -85,B 0,C 180,E1 -6169.953,E2 -6169.953} C_VEL
LIN {X 0,Y 495.73,Z 50.731,A -85,B 0,C 180,E1 -6172.553,E2 -6172.553} C_VEL
LIN {X 0,Y 495.78,Z 50.727,A -85,B 0,C 180,E1 -6175.457,E2 -6175.457} C_VEL
LIN {X 0,Y 495.757,Z 50.728,A -85,B 0,C 180,E1 -6178.364,E2 -6178.364} C_VEL
LIN {X 0,Y 495.79,Z 50.733,A -85,B 0,C 180,E1 -6181.507,E2 -6181.507} C_VEL
LIN {X 0,Y 495.84,Z 50.743,A -85,B 0,C 180,E1 -6184.028,E2 -6184.028} C_VEL
LIN {X 0,Y 497.582,Z 60.135,A -85,B 0,C 180,E1 -6185.598,E2 -6185.598} C_VEL
LIN {X 0,Y 497.314,Z 72.732,A -85,B 0,C 180,E1 -6187.569,E2 -6187.569} C_VEL
LIN {X 0,Y 496.785,Z 90.848,A -85,B 0,C 180,E1 -6190.367,E2 -6190.367} C_VEL
LIN {X 0,Y 496.314,Z 107.502,A -85,B 0,C 180,E1 -6192.912,E2 -6192.912} C_VEL
LIN {X 0,Y 496.152,Z 114.608,A -85,B 0,C 180,E1 -6193.98,E2 -6193.98} C_VEL
LIN {X 0,Y 498.438,Z 132.192,A -85,B 0,C 180,E1 -6194.307,E2 -6194.307} C_VEL
LIN {X 0,Y 497.907,Z 223.443,A -85,B 0,C 180,E1 -6195.647,E2 -6195.647} C_VEL
LIN {X 0,Y 497.573,Z 236.693,A -85,B 0,C 180,E1 -6196.002,E2 -6196.002} C_VEL
LIN {X 0,Y 497.192,Z 249.435,A -85,B 0,C 180,E1 -6196.512,E2 -6196.512} C_VEL
LIN {X 0,Y 496.84,Z 261.085,A -85,B 0,C 180,E1 -6197.148,E2 -6197.148} C_VEL
LIN {X 0,Y 496.407,Z 272.464,A -85,B 0,C 180,E1 -6197.946,E2 -6197.946} C_VEL
LIN {X 0,Y 496.055,Z 282.997,A -85,B 0,C 180,E1 -6198.87,E2 -6198.87} C_VEL
LIN {X 0,Y 495.749,Z 291.608,A -85,B 0,C 180,E1 -6199.793,E2 -6199.793} C_VEL
LIN {X 0,Y 495.464,Z 299.553,A -85,B 0,C 180,E1 -6200.817,E2 -6200.817} C_VEL
LIN {X 0,Y 495.302,Z 307.32,A -85,B 0,C 180,E1 -6202.048,E2 -6202.048} C_VEL
LIN {X 0,Y 495.107,Z 314.467,A -85,B 0,C 180,E1 -6203.479,E2 -6203.479} C_VEL
LIN {X 0,Y 495.096,Z 319.228,A -85,B 0,C 180,E1 -6204.706,E2 -6204.706} C_VEL
LIN {X 0,Y 495.056,Z 322.861,A -85,B 0,C 180,E1 -6205.929,E2 -6205.929} C_VEL
LIN {X 0,Y 495.077,Z 324.737,A -85,B 0,C 180,E1 -6206.745,E2 -6206.745} C_VEL
LIN {X 0,Y 495.062,Z 326.142,A -85,B 0,C 180,E1 -6207.559,E2 -6207.559} C_VEL
LIN {X 0,Y 494.934,Z 327.745,A -85,B 0,C 180,E1 -6209.186,E2 -6209.186} C_VEL
LIN {X 0,Y 494.933,Z 327.96,A -85,B 0,C 180,E1 -6210,E2 -6210} C_VEL
LIN {X 0,Y 494.97,Z 327.126,A -85,B 0,C 180,E1 -6211.627,E2 -6211.627} C_VEL
LIN {X 0,Y 495.062,Z 326.124,A -85,B 0,C 180,E1 -6212.441,E2 -6212.441} C_VEL
LIN {X 0,Y 495.077,Z 324.715,A -85,B 0,C 180,E1 -6213.255,E2 -6213.255} C_VEL
LIN {X 0,Y 495.007,Z 321.748,A -85,B 0,C 180,E1 -6214.478,E2 -6214.478} C_VEL
LIN {X 0,Y 495.075,Z 317.745,A -85,B 0,C 180,E1 -6215.703,E2 -6215.703} C_VEL
LIN {X 0,Y 495.192,Z 311.594,A -85,B 0,C 180,E1 -6217.133,E2 -6217.133} C_VEL
LIN {X 0,Y 495.338,Z 304.878,A -85,B 0,C 180,E1 -6218.362,E2 -6218.362} C_VEL
LIN {X 0,Y 495.589,Z 296.553,A -85,B 0,C 180,E1 -6219.591,E2 -6219.591} C_VEL
LIN {X 0,Y 495.925,Z 288.033,A -85,B 0,C 180,E1 -6220.616,E2 -6220.616} C_VEL
LIN {X 0,Y 496.324,Z 277.522,A -85,B 0,C 180,E1 -6221.641,E2 -6221.641} C_VEL
LIN {X 0,Y 496.597,Z 267.425,A -85,B 0,C 180,E1 -6222.443,E2 -6222.443} C_VEL
LIN {X 0,Y 497.047,Z 255.774,A -85,B 0,C 180,E1 -6223.179,E2 -6223.179} C_VEL
LIN {X 0,Y 497.39,Z 244.169,A -85,B 0,C 180,E1 -6223.742,E2 -6223.742} C_VEL
LIN {X 0,Y 497.757,Z 230.839,A -85,B 0,C 180,E1 -6224.201,E2 -6224.201} C_VEL
LIN {X 0,Y 498.045,Z 217.843,A -85,B 0,C 180,E1 -6224.479,E2 -6224.479} C_VEL
LIN {X 0,Y 498.474,Z 130.574,A -85,B 0,C 180,E1 -6225.753,E2 -6225.753} C_VEL
LIN {X 0,Y 496.181,Z 114.261,A -85,B 0,C 180,E1 -6226.075,E2 -6226.075} C_VEL
LIN {X 0,Y 496.786,Z 93.907,A -85,B 0,C 180,E1 -6229.203,E2 -6229.203} C_VEL
LIN {X 0,Y 497.333,Z 74.655,A -85,B 0,C 180,E1 -6232.21,E2 -6232.21} C_VEL
LIN {X 0,Y 497.791,Z 60.923,A -85,B 0,C 180,E1 -6234.391,E2 -6234.391} C_VEL
LIN {X 0,Y 495.823,Z 50.726,A -85,B 0,C 180,E1 -6236.168,E2 -6236.168} C_VEL
LIN {X 0,Y 495.773,Z 50.731,A -85,B 0,C 180,E1 -6238.814,E2 -6238.814} C_VEL
LIN {X 0,Y 495.755,Z 50.734,A -85,B 0,C 180,E1 -6241.725,E2 -6241.725} C_VEL
LIN {X 0,Y 495.77,Z 50.726,A -85,B 0,C 180,E1 -6244.694,E2 -6244.694} C_VEL
LIN {X 0,Y 495.731,Z 50.735,A -85,B 0,C 180,E1 -6247.561,E2 -6247.561} C_VEL
LIN {X 0,Y 495.765,Z 50.727,A -85,B 0,C 180,E1 -6250.7,E2 -6250.7} C_VEL
LIN {X 0,Y 495.727,Z 50.733,A -85,B 0,C 180,E1 -6254.001,E2 -6254.001} C_VEL
LIN {X 0,Y 495.724,Z 50.732,A -85,B 0,C 180,E1 -6257.117,E2 -6257.117} C_VEL
LIN {X 0,Y 495.788,Z 50.725,A -85,B 0,C 180,E1 -6259.948,E2 -6259.948} C_VEL
LIN {X 0,Y 495.729,Z 50.729,A -85,B 0,C 180,E1 -6262.552,E2 -6262.552} C_VEL
LIN {X 0,Y 495.784,Z 50.727,A -85,B 0,C 180,E1 -6265.457,E2 -6265.457} C_VEL
LIN {X 0,Y 495.754,Z 50.729,A -85,B 0,C 180,E1 -6268.364,E2 -6268.364} C_VEL
LIN {X 0,Y 495.786,Z 50.725,A -85,B 0,C 180,E1 -6271.507,E2 -6271.507} C_VEL
LIN {X 0,Y 495.789,Z 50.721,A -85,B 0,C 180,E1 -6273.932,E2 -6273.932} C_VEL
LIN {X 0,Y 495.763,Z 50.725,A -85,B 0,C 180,E1 -6277.137,E2 -6277.137} C_VEL
LIN {X 0,Y 495.776,Z 50.727,A -85,B 0,C 180,E1 -6280.11,E2 -6280.11} C_VEL
LIN {X 0,Y 495.785,Z 50.728,A -85,B 0,C 180,E1 -6282.681,E2 -6282.681} C_VEL
LIN {X 0,Y 495.788,Z 50.723,A -85,B 0,C 180,E1 -6285.217,E2 -6285.217} C_VEL
LIN {X 0,Y 495.85,Z 50.72,A -85,B 0,C 180,E1 -6288.555,E2 -6288.555} C_VEL
LIN {X 0,Y 495.871,Z 50.717,A -85,B 0,C 180,E1 -6291.852,E2 -6291.852} C_VEL
LIN {X 0,Y 495.889,Z 50.715,A -85,B 0,C 180,E1 -6294.307,E2 -6294.307} C_VEL
LIN {X 0,Y 495.99,Z 50.7,A -85,B 0,C 180,E1 -6297.564,E2 -6297.564} C_VEL
LIN {X 0,Y 495.995,Z 50.702,A -85,B 0,C 180,E1 -6300,E2 -6300} C_VEL
LIN {X 0,Y 495.989,Z 50.695,A -85,B 0,C 180,E1 -6302.437,E2 -6302.437} C_VEL
LIN {X 0,Y 495.885,Z 50.716,A -85,B 0,C 180,E1 -6305.694,E2 -6305.694} C_VEL
LIN {X 0,Y 495.834,Z 50.714,A -85,B 0,C 180,E1 -6308.149,E2 -6308.149} C_VEL
LIN {X 0,Y 495.849,Z 50.719,A -85,B 0,C 180,E1 -6311.446,E2 -6311.446} C_VEL
LIN {X 0,Y 495.788,Z 50.726,A -85,B 0,C 180,E1 -6314.783,E2 -6314.783} C_VEL
LIN {X 0,Y 495.763,Z 50.728,A -85,B 0,C 180,E1 -6317.32,E2 -6317.32} C_VEL
LIN {X 0,Y 495.769,Z 50.726,A -85,B 0,C 180,E1 -6319.891,E2 -6319.891} C_VEL
LIN {X 0,Y 495.758,Z 50.734,A -85,B 0,C 180,E1 -6322.861,E2 -6322.861} C_VEL
LIN {X 0,Y 495.758,Z 50.726,A -85,B 0,C 180,E1 -6326.07,E2 -6326.07} C_VEL
LIN {X 0,Y 495.743,Z 50.732,A -85,B 0,C 180,E1 -6328.817,E2 -6328.817} C_VEL
LIN {X 0,Y 495.754,Z 50.729,A -85,B 0,C 180,E1 -6331.726,E2 -6331.726} C_VEL
LIN {X 0,Y 495.76,Z 50.728,A -85,B 0,C 180,E1 -6334.693,E2 -6334.693} C_VEL
LIN {X 0,Y 495.72,Z 50.734,A -85,B 0,C 180,E1 -6337.563,E2 -6337.563} C_VEL
LIN {X 0,Y 495.743,Z 50.735,A -85,B 0,C 180,E1 -6340.045,E2 -6340.045} C_VEL
LIN {X 0,Y 495.703,Z 50.738,A -85,B 0,C 180,E1 -6342.886,E2 -6342.886} C_VEL
LIN {X 0,Y 495.723,Z 50.741,A -85,B 0,C 180,E1 -6345.998,E2 -6345.998} C_VEL
LIN {X 0,Y 495.731,Z 50.735,A -85,B 0,C 180,E1 -6349.297,E2 -6349.297} C_VEL
LIN {X 0,Y 495.725,Z 50.738,A -85,B 0,C 180,E1 -6351.407,E2 -6351.407} C_VEL
LIN {X 0,Y 495.744,Z 50.733,A -85,B 0,C 180,E1 -6354.462,E2 -6354.462} C_VEL
LIN {X 0,Y 495.786,Z 50.774,A -85,B 0,C 180,E1 -6356.974,E2 -6356.974} C_VEL
LIN {X 0,Y 496.614,Z 55.875,A -85,B 0,C 180,E1 -6358.116,E2 -6358.116} C_VEL
LIN {X 0,Y 496.555,Z 61.452,A -85,B 0,C 180,E1 -6359.298,E2 -6359.298} C_VEL
LIN {X 0,Y 496.138,Z 63.532,A -85,B 0,C 180,E1 -6359.581,E2 -6359.581} C_VEL
LIN {X 0,Y 494.965,Z 67.075,A -85,B 0,C 180,E1 -6359.816,E2 -6359.816} C_VEL
LIN {X 0,Y 493.158,Z 72.615,A -85,B 0,C 180,E1 -6359.978,E2 -6359.978} C_VEL
LIN {X 0,Y 492.135,Z 79.286,A -85,B 0,C 180,E1 -6360.06,E2 -6360.06} C_VEL
LIN {X 0,Y 491.932,Z 91.695,A -85,B 0,C 180,E1 -6360.239,E2 -6360.239} C_VEL
LIN {X 0,Y 491.273,Z 172.18,A -85,B 0,C 180,E1 -6361.452,E2 -6361.452} C_VEL
LIN {X 0,Y 491.107,Z 186.002,A -85,B 0,C 180,E1 -6361.849,E2 -6361.849} C_VEL
LIN {X 0,Y 490.837,Z 197.473,A -85,B 0,C 180,E1 -6362.332,E2 -6362.332} C_VEL
LIN {X 0,Y 490.484,Z 208.417,A -85,B 0,C 180,E1 -6362.94,E2 -6362.94} C_VEL
LIN {X 0,Y 490.031,Z 219.372,A -85,B 0,C 180,E1 -6363.717,E2 -6363.717} C_VEL
LIN {X 0,Y 489.655,Z 230.568,A -85,B 0,C 180,E1 -6364.722,E2 -6364.722} C_VEL
LIN {X 0,Y 489.243,Z 240.473,A -85,B 0,C 180,E1 -6365.833,E2 -6365.833} C_VEL
LIN {X 0,Y 488.896,Z 248.398,A -85,B 0,C 180,E1 -6366.93,E2 -6366.93} C_VEL
LIN {X 0,Y 488.559,Z 256.17,A -85,B 0,C 180,E1 -6368.259,E2 -6368.259} C_VEL
LIN {X 0,Y 488.39,Z 262.095,A -85,B 0,C 180,E1 -6369.537,E2 -6369.537} C_VEL
LIN {X 0,Y 488.231,Z 266.242,A -85,B 0,C 180,E1 -6370.666,E2 -6370.666} C_VEL
LIN {X 0,Y 488.083,Z 269.69,A -85,B 0,C 180,E1 -6371.87,E2 -6371.87} C_VEL
LIN {X 0,Y 487.949,Z 272.519,A -85,B 0,C 180,E1 -6373.258,E2 -6373.258} C_VEL
LIN {X 0,Y 487.923,Z 274.298,A -85,B 0,C 180,E1 -6374.812,E2 -6374.812} C_VEL
LIN {X 0,Y 487.916,Z 274.695,A -85,B 0,C 180,E1 -6375.826,E2 -6375.826} C_VEL
LIN {X 0,Y 487.934,Z 274.599,A -85,B 0,C 180,E1 -6376.676,E2 -6376.676} C_VEL
LIN {X 0,Y 488.003,Z 273.159,A -85,B 0,C 180,E1 -6378.326,E2 -6378.326} C_VEL
LIN {X 0,Y 488.033,Z 271.755,A -85,B 0,C 180,E1 -6379.21,E2 -6379.21} C_VEL
LIN {X 0,Y 488.098,Z 268.906,A -85,B 0,C 180,E1 -6380.469,E2 -6380.469} C_VEL
LIN {X 0,Y 488.229,Z 265.025,A -85,B 0,C 180,E1 -6381.724,E2 -6381.724} C_VEL
LIN {X 0,Y 488.42,Z 259.208,A -85,B 0,C 180,E1 -6383.152,E2 -6383.152} C_VEL
LIN {X 0,Y 488.66,Z 252.521,A -85,B 0,C 180,E1 -6384.429,E2 -6384.429} C_VEL
LIN {X 0,Y 488.963,Z 244.414,A -85,B 0,C 180,E1 -6385.673,E2 -6385.673} C_VEL
LIN {X 0,Y 489.312,Z 236.13,A -85,B 0,C 180,E1 -6386.707,E2 -6386.707} C_VEL
LIN {X 0,Y 489.732,Z 225.947,A -85,B 0,C 180,E1 -6387.739,E2 -6387.739} C_VEL
LIN {X 0,Y 490.171,Z 214.474,A -85,B 0,C 180,E1 -6388.665,E2 -6388.665} C_VEL
LIN {X 0,Y 490.538,Z 203.18,A -85,B 0,C 180,E1 -6389.385,E2 -6389.385} C_VEL
LIN {X 0,Y 490.83,Z 190.3,A -85,B 0,C 180,E1 -6390,E2 -6390} C_VEL
LIN {X 0,Y 491.027,Z 178.26,A -85,B 0,C 180,E1 -6390.41,E2 -6390.41} C_VEL
LIN {X 0,Y 491.203,Z 164.964,A -85,B 0,C 180,E1 -6390.692,E2 -6390.692} C_VEL
LIN {X 0,Y 491.719,Z 76.189,A -85,B 0,C 180,E1 -6391.997,E2 -6391.997} C_VEL
LIN {X 0,Y 489.359,Z 64.753,A -85,B 0,C 180,E1 -6392.264,E2 -6392.264} C_VEL
LIN {X 0,Y 489.477,Z 55.992,A -85,B 0,C 180,E1 -6394.117,E2 -6394.117} C_VEL
LIN {X 0,Y 488.831,Z 51.598,A -85,B 0,C 180,E1 -6395.104,E2 -6395.104} C_VEL
LIN {X 0,Y 488.869,Z 51.588,A -85,B 0,C 180,E1 -6397.434,E2 -6397.434} C_VEL
LIN {X 0,Y 488.742,Z 51.606,A -85,B 0,C 180,E1 -6400.774,E2 -6400.774} C_VEL
LIN {X 0,Y 488.736,Z 51.602,A -85,B 0,C 180,E1 -6403.302,E2 -6403.302} C_VEL
LIN {X 0,Y 488.767,Z 51.599,A -85,B 0,C 180,E1 -6405.855,E2 -6405.855} C_VEL
LIN {X 0,Y 488.748,Z 51.6,A -85,B 0,C 180,E1 -6409.313,E2 -6409.313} C_VEL
LIN {X 0,Y 488.704,Z 51.611,A -85,B 0,C 180,E1 -6411.957,E2 -6411.957} C_VEL
LIN {X 0,Y 488.724,Z 51.603,A -85,B 0,C 180,E1 -6415.046,E2 -6415.046} C_VEL
LIN {X 0,Y 488.751,Z 51.601,A -85,B 0,C 180,E1 -6417.397,E2 -6417.397} C_VEL
LIN {X 0,Y 488.715,Z 51.606,A -85,B 0,C 180,E1 -6420.363,E2 -6420.363} C_VEL
LIN {X 0,Y 488.741,Z 51.605,A -85,B 0,C 180,E1 -6423.484,E2 -6423.484} C_VEL
LIN {X 0,Y 488.692,Z 51.608,A -85,B 0,C 180,E1 -6426.355,E2 -6426.355} C_VEL
LIN {X 0,Y 488.705,Z 51.609,A -85,B 0,C 180,E1 -6429.254,E2 -6429.254} C_VEL
LIN {X 0,Y 488.712,Z 51.611,A -85,B 0,C 180,E1 -6431.6,E2 -6431.6} C_VEL
LIN {X 0,Y 488.705,Z 51.607,A -85,B 0,C 180,E1 -6434.802,E2 -6434.802} C_VEL
LIN {X 0,Y 488.696,Z 51.612,A -85,B 0,C 180,E1 -6437.474,E2 -6437.474} C_VEL
LIN {X 0,Y 488.737,Z 51.604,A -85,B 0,C 180,E1 -6439.676,E2 -6439.676} C_VEL
LIN {X 0,Y 488.683,Z 51.613,A -85,B 0,C 180,E1 -6442.841,E2 -6442.841} C_VEL
LIN {X 0,Y 488.735,Z 51.602,A -85,B 0,C 180,E1 -6445.887,E2 -6445.887} C_VEL
LIN {X 0,Y 488.696,Z 51.614,A -85,B 0,C 180,E1 -6448.82,E2 -6448.82} C_VEL
LIN {X 0,Y 488.748,Z 51.6,A -85,B 0,C 180,E1 -6451.671,E2 -6451.671} C_VEL
LIN {X 0,Y 488.751,Z 51.604,A -85,B 0,C 180,E1 -6454.444,E2 -6454.444} C_VEL
LIN {X 0,Y 488.727,Z 51.604,A -85,B 0,C 180,E1 -6457.153,E2 -6457.153} C_VEL
LIN {X 0,Y 488.728,Z 51.603,A -85,B 0,C 180,E1 -6459.81,E2 -6459.81} C_VEL
LIN {X 0,Y 488.733,Z 51.61,A -85,B 0,C 180,E1 -6462.423,E2 -6462.423} C_VEL
LIN {X 0,Y 488.765,Z 51.599,A -85,B 0,C 180,E1 -6464.999,E2 -6464.999} C_VEL
LIN {X 0,Y 488.809,Z 51.598,A -85,B 0,C 180,E1 -6468.387,E2 -6468.387} C_VEL
LIN {X 0,Y 488.819,Z 51.595,A -85,B 0,C 180,E1 -6471.733,E2 -6471.733} C_VEL
LIN {X 0,Y 488.852,Z 51.592,A -85,B 0,C 180,E1 -6474.224,E2 -6474.224} C_VEL
LIN {X 0,Y 488.962,Z 51.577,A -85,B 0,C 180,E1 -6477.528,E2 -6477.528} C_VEL
LIN {X 0,Y 488.936,Z 51.576,A -85,B 0,C 180,E1 -6480.823,E2 -6480.823} C_VEL
LIN {X 0,Y 488.961,Z 51.574,A -85,B 0,C 180,E1 -6482.471,E2 -6482.471} C_VEL
LIN {X 0,Y 488.848,Z 51.593,A -85,B 0,C 180,E1 -6485.776,E2 -6485.776} C_VEL
LIN {X 0,Y 488.788,Z 51.595,A -85,B 0,C 180,E1 -6488.267,E2 -6488.267} C_VEL
LIN {X 0,Y 488.807,Z 51.598,A -85,B 0,C 180,E1 -6491.612,E2 -6491.612} C_VEL
LIN {X 0,Y 488.764,Z 51.603,A -85,B 0,C 180,E1 -6495,E2 -6495} C_VEL
LIN {X 0,Y 488.749,Z 51.601,A -85,B 0,C 180,E1 -6498.442,E2 -6498.442} C_VEL
LIN {X 0,Y 488.709,Z 51.613,A -85,B 0,C 180,E1 -6501.071,E2 -6501.071} C_VEL
LIN {X 0,Y 488.689,Z 51.608,A -85,B 0,C 180,E1 -6503.746,E2 -6503.746} C_VEL
LIN {X 0,Y 488.739,Z 51.604,A -85,B 0,C 180,E1 -6506.473,E2 -6506.473} C_VEL
LIN {X 0,Y 488.724,Z 51.605,A -85,B 0,C 180,E1 -6509.27,E2 -6509.27} C_VEL
LIN {X 0,Y 488.705,Z 51.607,A -85,B 0,C 180,E1 -6512.147,E2 -6512.147} C_VEL
LIN {X 0,Y 488.719,Z 51.605,A -85,B 0,C 180,E1 -6515.115,E2 -6515.115} C_VEL
LIN {X 0,Y 488.681,Z 51.613,A -85,B 0,C 180,E1 -6518.2,E2 -6518.2} C_VEL
LIN {X 0,Y 488.72,Z 51.611,A -85,B 0,C 180,E1 -6520.345,E2 -6520.345} C_VEL
LIN {X 0,Y 488.686,Z 51.609,A -85,B 0,C 180,E1 -6523.655,E2 -6523.655} C_VEL
LIN {X 0,Y 488.686,Z 51.613,A -85,B 0,C 180,E1 -6526.345,E2 -6526.345} C_VEL
LIN {X 0,Y 488.735,Z 51.605,A -85,B 0,C 180,E1 -6529.677,E2 -6529.677} C_VEL
LIN {X 0,Y 488.681,Z 51.608,A -85,B 0,C 180,E1 -6532.841,E2 -6532.841} C_VEL
LIN {X 0,Y 488.733,Z 51.609,A -85,B 0,C 180,E1 -6535.887,E2 -6535.887} C_VEL
LIN {X 0,Y 488.693,Z 51.607,A -85,B 0,C 180,E1 -6538.82,E2 -6538.82} C_VEL
LIN {X 0,Y 488.746,Z 51.61,A -85,B 0,C 180,E1 -6541.671,E2 -6541.671} C_VEL
LIN {X 0,Y 488.811,Z 51.725,A -85,B 0,C 180,E1 -6543.876,E2 -6543.876} C_VEL
LIN {X 0,Y 490.586,Z 61.013,A -85,B 0,C 180,E1 -6545.452,E2 -6545.452} C_VEL
LIN {X 0,Y 490.47,Z 70.955,A -85,B 0,C 180,E1 -6547.036,E2 -6547.036} C_VEL
LIN {X 0,Y 489.861,Z 88.967,A -85,B 0,C 180,E1 -6549.859,E2 -6549.859} C_VEL
LIN {X 0,Y 489.326,Z 107.024,A -85,B 0,C 180,E1 -6552.661,E2 -6552.661} C_VEL
LIN {X 0,Y 489.158,Z 114.09,A -85,B 0,C 180,E1 -6553.751,E2 -6553.751} C_VEL
LIN {X 0,Y 491.553,Z 131.436,A -85,B 0,C 180,E1 -6554.091,E2 -6554.091} C_VEL
LIN {X 0,Y 491.001,Z 223.666,A -85,B 0,C 180,E1 -6555.467,E2 -6555.467} C_VEL
LIN {X 0,Y 490.649,Z 236.724,A -85,B 0,C 180,E1 -6555.827,E2 -6555.827} C_VEL
LIN {X 0,Y 490.285,Z 248.8,A -85,B 0,C 180,E1 -6556.319,E2 -6556.319} C_VEL
LIN {X 0,Y 489.888,Z 260.525,A -85,B 0,C 180,E1 -6556.962,E2 -6556.962} C_VEL
LIN {X 0,Y 489.435,Z 272,A -85,B 0,C 180,E1 -6557.776,E2 -6557.776} C_VEL
LIN {X 0,Y 489.062,Z 282.509,A -85,B 0,C 180,E1 -6558.708,E2 -6558.708} C_VEL
LIN {X 0,Y 488.701,Z 291.142,A -85,B 0,C 180,E1 -6559.644,E2 -6559.644} C_VEL
LIN {X 0,Y 488.425,Z 299.108,A -85,B 0,C 180,E1 -6560.684,E2 -6560.684} C_VEL
LIN {X 0,Y 488.228,Z 306.894,A -85,B 0,C 180,E1 -6561.932,E2 -6561.932} C_VEL
LIN {X 0,Y 488.036,Z 314.053,A -85,B 0,C 180,E1 -6563.384,E2 -6563.384} C_VEL
LIN {X 0,Y 488.001,Z 318.821,A -85,B 0,C 180,E1 -6564.628,E2 -6564.628} C_VEL
LIN {X 0,Y 487.95,Z 322.461,A -85,B 0,C 180,E1 -6565.87,E2 -6565.87} C_VEL
LIN {X 0,Y 487.997,Z 324.343,A -85,B 0,C 180,E1 -6566.697,E2 -6566.697} C_VEL
LIN {X 0,Y 487.968,Z 325.75,A -85,B 0,C 180,E1 -6567.523,E2 -6567.523} C_VEL
LIN {X 0,Y 487.856,Z 327.358,A -85,B 0,C 180,E1 -6569.174,E2 -6569.174} C_VEL
LIN {X 0,Y 487.852,Z 327.576,A -85,B 0,C 180,E1 -6570,E2 -6570} C_VEL
LIN {X 0,Y 487.899,Z 326.746,A -85,B 0,C 180,E1 -6571.651,E2 -6571.651} C_VEL
LIN {X 0,Y 487.968,Z 325.745,A -85,B 0,C 180,E1 -6572.476,E2 -6572.476} C_VEL
LIN {X 0,Y 487.997,Z 324.339,A -85,B 0,C 180,E1 -6573.302,E2 -6573.302} C_VEL
LIN {X 0,Y 487.92,Z 321.376,A -85,B 0,C 180,E1 -6574.544,E2 -6574.544} C_VEL
LIN {X 0,Y 487.973,Z 317.377,A -85,B 0,C 180,E1 -6575.786,E2 -6575.786} C_VEL
LIN {X 0,Y 488.112,Z 311.238,A -85,B 0,C 180,E1 -6577.237,E2 -6577.237} C_VEL
LIN {X 0,Y 488.285,Z 304.534,A -85,B 0,C 180,E1 -6578.484,E2 -6578.484} C_VEL
LIN {X 0,Y 488.519,Z 296.223,A -85,B 0,C 180,E1 -6579.732,E2 -6579.732} C_VEL
LIN {X 0,Y 488.921,Z 287.728,A -85,B 0,C 180,E1 -6580.77,E2 -6580.77} C_VEL
LIN {X 0,Y 489.326,Z 277.311,A -85,B 0,C 180,E1 -6581.804,E2 -6581.804} C_VEL
LIN {X 0,Y 489.708,Z 266.11,A -85,B 0,C 180,E1 -6582.7,E2 -6582.7} C_VEL
LIN {X 0,Y 490.142,Z 253.697,A -85,B 0,C 180,E1 -6583.474,E2 -6583.474} C_VEL
LIN {X 0,Y 490.567,Z 241.486,A -85,B 0,C 180,E1 -6584.043,E2 -6584.043} C_VEL
LIN {X 0,Y 490.982,Z 228.156,A -85,B 0,C 180,E1 -6584.48,E2 -6584.48} C_VEL
LIN {X 0,Y 491.182,Z 213.142,A -85,B 0,C 180,E1 -6584.765,E2 -6584.765} C_VEL
LIN {X 0,Y 491.677,Z 131.209,A -85,B 0,C 180,E1 -6585.976,E2 -6585.976} C_VEL
LIN {X 0,Y 489.19,Z 113.789,A -85,B 0,C 180,E1 -6586.338,E2 -6586.338} C_VEL
LIN {X 0,Y 489.844,Z 93.662,A -85,B 0,C 180,E1 -6589.486,E2 -6589.486} C_VEL
LIN {X 0,Y 490.457,Z 74.443,A -85,B 0,C 180,E1 -6592.539,E2 -6592.539} C_VEL
LIN {X 0,Y 490.858,Z 62.103,A -85,B 0,C 180,E1 -6594.533,E2 -6594.533} C_VEL
LIN {X 0,Y 488.813,Z 51.598,A -85,B 0,C 180,E1 -6596.411,E2 -6596.411} C_VEL
LIN {X 0,Y 488.724,Z 51.608,A -85,B 0,C 180,E1 -6599.27,E2 -6599.27} C_VEL
LIN {X 0,Y 488.702,Z 51.614,A -85,B 0,C 180,E1 -6602.147,E2 -6602.147} C_VEL
LIN {X 0,Y 488.721,Z 51.603,A -85,B 0,C 180,E1 -6605.114,E2 -6605.114} C_VEL
LIN {X 0,Y 488.68,Z 51.614,A -85,B 0,C 180,E1 -6608.2,E2 -6608.2} C_VEL
LIN {X 0,Y 488.717,Z 51.607,A -85,B 0,C 180,E1 -6610.344,E2 -6610.344} C_VEL
LIN {X 0,Y 488.683,Z 51.616,A -85,B 0,C 180,E1 -6613.654,E2 -6613.654} C_VEL
LIN {X 0,Y 488.682,Z 51.607,A -85,B 0,C 180,E1 -6616.345,E2 -6616.345} C_VEL
LIN {X 0,Y 488.732,Z 51.607,A -85,B 0,C 180,E1 -6619.676,E2 -6619.676} C_VEL
LIN {X 0,Y 488.678,Z 51.607,A -85,B 0,C 180,E1 -6622.277,E2 -6622.277} C_VEL
LIN {X 0,Y 488.727,Z 51.609,A -85,B 0,C 180,E1 -6625.051,E2 -6625.051} C_VEL
LIN {X 0,Y 488.702,Z 51.606,A -85,B 0,C 180,E1 -6628.046,E2 -6628.046} C_VEL
LIN {X 0,Y 488.721,Z 51.607,A -85,B 0,C 180,E1 -6630.73,E2 -6630.73} C_VEL
LIN {X 0,Y 488.755,Z 51.598,A -85,B 0,C 180,E1 -6633.528,E2 -6633.528} C_VEL
LIN {X 0,Y 488.691,Z 51.61,A -85,B 0,C 180,E1 -6636.255,E2 -6636.255} C_VEL
LIN {X 0,Y 488.744,Z 51.603,A -85,B 0,C 180,E1 -6639.176,E2 -6639.176} C_VEL
LIN {X 0,Y 488.757,Z 51.597,A -85,B 0,C 180,E1 -6641.628,E2 -6641.628} C_VEL
LIN {X 0,Y 488.76,Z 51.6,A -85,B 0,C 180,E1 -6645,E2 -6645} C_VEL
LIN {X 0,Y 488.803,Z 51.6,A -85,B 0,C 180,E1 -6648.388,E2 -6648.388} C_VEL
LIN {X 0,Y 488.815,Z 51.594,A -85,B 0,C 180,E1 -6651.734,E2 -6651.734} C_VEL
LIN {X 0,Y 488.848,Z 51.593,A -85,B 0,C 180,E1 -6654.224,E2 -6654.224} C_VEL
LIN {X 0,Y 488.958,Z 51.576,A -85,B 0,C 180,E1 -6657.529,E2 -6657.529} C_VEL
LIN {X 0,Y 488.966,Z 51.578,A -85,B 0,C 180,E1 -6660,E2 -6660} C_VEL
LIN {X 0,Y 488.957,Z 51.57,A -85,B 0,C 180,E1 -6662.472,E2 -6662.472} C_VEL
LIN {X 0,Y 488.844,Z 51.592,A -85,B 0,C 180,E1 -6665.776,E2 -6665.776} C_VEL
LIN {X 0,Y 488.783,Z 51.592,A -85,B 0,C 180,E1 -6668.267,E2 -6668.267} C_VEL
LIN {X 0,Y 488.803,Z 51.595,A -85,B 0,C 180,E1 -6671.613,E2 -6671.613} C_VEL
LIN {X 0,Y 488.76,Z 51.605,A -85,B 0,C 180,E1 -6675.001,E2 -6675.001} C_VEL
LIN {X 0,Y 488.745,Z 51.6,A -85,B 0,C 180,E1 -6678.443,E2 -6678.443} C_VEL
LIN {X 0,Y 488.705,Z 51.607,A -85,B 0,C 180,E1 -6681.071,E2 -6681.071} C_VEL
LIN {X 0,Y 488.682,Z 51.609,A -85,B 0,C 180,E1 -6683.746,E2 -6683.746} C_VEL
LIN {X 0,Y 488.723,Z 51.608,A -85,B 0,C 180,E1 -6686.929,E2 -6686.929} C_VEL
LIN {X 0,Y 488.723,Z 51.607,A -85,B 0,C 180,E1 -6690.22,E2 -6690.22} C_VEL
LIN {X 0,Y 488.728,Z 51.603,A -85,B 0,C 180,E1 -6693.484,E2 -6693.484} C_VEL
LIN {X 0,Y 488.672,Z 51.617,A -85,B 0,C 180,E1 -6696.354,E2 -6696.354} C_VEL
LIN {X 0,Y 488.693,Z 51.61,A -85,B 0,C 180,E1 -6699.256,E2 -6699.256} C_VEL
LIN {X 0,Y 488.666,Z 51.616,A -85,B 0,C 180,E1 -6702.529,E2 -6702.529} C_VEL
LIN {X 0,Y 488.701,Z 51.607,A -85,B 0,C 180,E1 -6705.198,E2 -6705.198} C_VEL
LIN {X 0,Y 488.676,Z 51.61,A -85,B 0,C 180,E1 -6708.582,E2 -6708.582} C_VEL
LIN {X 0,Y 488.689,Z 51.611,A -85,B 0,C 180,E1 -6710.95,E2 -6710.95} C_VEL
LIN {X 0,Y 488.667,Z 51.618,A -85,B 0,C 180,E1 -6713.867,E2 -6713.867} C_VEL
LIN {X 0,Y 488.741,Z 51.65,A -85,B 0,C 180,E1 -6716.788,E2 -6716.788} C_VEL
LIN {X 0,Y 489.702,Z 57.77,A -85,B 0,C 180,E1 -6718.169,E2 -6718.169} C_VEL
LIN {X 0,Y 489.554,Z 65.085,A -85,B 0,C 180,E1 -6719.739,E2 -6719.739} C_VEL
LIN {X 0,Y 491.96,Z 76.226,A -85,B 0,C 180,E1 -6720.007,E2 -6720.007} C_VEL
LIN {X 0,Y 491.932,Z 91.695,A -85,B 0,C 180,E1 -6720.239,E2 -6720.239} C_VEL
LIN {X 0,Y 491.202,Z 97.541,A -85,B 0,C 180,E1 -6720.3,E2 -6720.3} C_VEL
LIN {X 0,Y 485.593,Z 116.553,A -85,B 0,C 180,E1 -6720.382,E2 -6720.382} C_VEL
LIN {X 0,Y 484.949,Z 122.395,A -85,B 0,C 180,E1 -6720.448,E2 -6720.448} C_VEL
LIN {X 0,Y 484.474,Z 172.522,A -85,B 0,C 180,E1 -6721.221,E2 -6721.221} C_VEL
LIN {X 0,Y 484.292,Z 186.356,A -85,B 0,C 180,E1 -6721.624,E2 -6721.624} C_VEL
LIN {X 0,Y 484.002,Z 198.308,A -85,B 0,C 180,E1 -6722.136,E2 -6722.136} C_VEL
LIN {X 0,Y 483.613,Z 209.414,A -85,B 0,C 180,E1 -6722.771,E2 -6722.771} C_VEL
LIN {X 0,Y 483.12,Z 220.071,A -85,B 0,C 180,E1 -6723.545,E2 -6723.545} C_VEL
LIN {X 0,Y 482.755,Z 230.596,A -85,B 0,C 180,E1 -6724.503,E2 -6724.503} C_VEL
LIN {X 0,Y 482.356,Z 239.24,A -85,B 0,C 180,E1 -6725.465,E2 -6725.465} C_VEL
LIN {X 0,Y 481.96,Z 247.698,A -85,B 0,C 180,E1 -6726.61,E2 -6726.61} C_VEL
LIN {X 0,Y 481.589,Z 255.501,A -85,B 0,C 180,E1 -6727.928,E2 -6727.928} C_VEL
LIN {X 0,Y 481.389,Z 261.213,A -85,B 0,C 180,E1 -6729.127,E2 -6729.127} C_VEL
LIN {X 0,Y 481.212,Z 265.959,A -85,B 0,C 180,E1 -6730.372,E2 -6730.372} C_VEL
LIN {X 0,Y 481.021,Z 269.963,A -85,B 0,C 180,E1 -6731.75,E2 -6731.75} C_VEL
LIN {X 0,Y 480.878,Z 272.567,A -85,B 0,C 180,E1 -6733.005,E2 -6733.005} C_VEL
LIN {X 0,Y 480.874,Z 273.837,A -85,B 0,C 180,E1 -6733.878,E2 -6733.878} C_VEL
LIN {X 0,Y 480.836,Z 274.664,A -85,B 0,C 180,E1 -6734.747,E2 -6734.747} C_VEL
LIN {X 0,Y 480.845,Z 275.043,A -85,B 0,C 180,E1 -6735.613,E2 -6735.613} C_VEL
LIN {X 0,Y 480.833,Z 275.026,A -85,B 0,C 180,E1 -6736.476,E2 -6736.476} C_VEL
LIN {X 0,Y 480.852,Z 274.611,A -85,B 0,C 180,E1 -6737.336,E2 -6737.336} C_VEL
LIN {X 0,Y 480.91,Z 273.635,A -85,B 0,C 180,E1 -6738.278,E2 -6738.278} C_VEL
LIN {X 0,Y 480.974,Z 270.797,A -85,B 0,C 180,E1 -6739.902,E2 -6739.902} C_VEL
LIN {X 0,Y 481.08,Z 267.426,A -85,B 0,C 180,E1 -6741.177,E2 -6741.177} C_VEL
LIN {X 0,Y 481.261,Z 262.974,A -85,B 0,C 180,E1 -6742.448,E2 -6742.448} C_VEL
LIN {X 0,Y 481.443,Z 257.339,A -85,B 0,C 180,E1 -6743.715,E2 -6743.715} C_VEL
LIN {X 0,Y 481.745,Z 250.272,A -85,B 0,C 180,E1 -6744.979,E2 -6744.979} C_VEL
LIN {X 0,Y 482.091,Z 241.494,A -85,B 0,C 180,E1 -6746.239,E2 -6746.239} C_VEL
LIN {X 0,Y 482.515,Z 232.49,A -85,B 0,C 180,E1 -6747.287,E2 -6747.287} C_VEL
LIN {X 0,Y 482.889,Z 222.576,A -85,B 0,C 180,E1 -6748.228,E2 -6748.228} C_VEL
LIN {X 0,Y 483.362,Z 211.535,A -85,B 0,C 180,E1 -6749.063,E2 -6749.063} C_VEL
LIN {X 0,Y 483.72,Z 199.235,A -85,B 0,C 180,E1 -6749.792,E2 -6749.792} C_VEL
LIN {X 0,Y 483.975,Z 186.795,A -85,B 0,C 180,E1 -6750.338,E2 -6750.338} C_VEL
LIN {X 0,Y 484.255,Z 173.543,A -85,B 0,C 180,E1 -6750.728,E2 -6750.728} C_VEL
LIN {X 0,Y 484.424,Z 151.476,A -85,B 0,C 180,E1 -6751.091,E2 -6751.091} C_VEL
LIN {X 0,Y 484.783,Z 76.768,A -85,B 0,C 180,E1 -6752.209,E2 -6752.209} C_VEL
LIN {X 0,Y 482.396,Z 65.116,A -85,B 0,C 180,E1 -6752.479,E2 -6752.479} C_VEL
LIN {X 0,Y 482.485,Z 57.163,A -85,B 0,C 180,E1 -6754.177,E2 -6754.177} C_VEL
LIN {X 0,Y 481.818,Z 52.47,A -85,B 0,C 180,E1 -6755.231,E2 -6755.231} C_VEL
LIN {X 0,Y 481.834,Z 52.464,A -85,B 0,C 180,E1 -6757.543,E2 -6757.543} C_VEL
LIN {X 0,Y 481.711,Z 52.48,A -85,B 0,C 180,E1 -6760.934,E2 -6760.934} C_VEL
LIN {X 0,Y 481.7,Z 52.478,A -85,B 0,C 180,E1 -6763.5,E2 -6763.5} C_VEL
LIN {X 0,Y 481.7,Z 52.482,A -85,B 0,C 180,E1 -6766.094,E2 -6766.094} C_VEL
LIN {X 0,Y 481.714,Z 52.479,A -85,B 0,C 180,E1 -6768.722,E2 -6768.722} C_VEL
LIN {X 0,Y 481.651,Z 52.484,A -85,B 0,C 180,E1 -6771.395,E2 -6771.395} C_VEL
LIN {X 0,Y 481.667,Z 52.49,A -85,B 0,C 180,E1 -6774.114,E2 -6774.114} C_VEL
LIN {X 0,Y 481.752,Z 52.472,A -85,B 0,C 180,E1 -6777.139,E2 -6777.139} C_VEL
LIN {X 0,Y 481.684,Z 52.486,A -85,B 0,C 180,E1 -6779.741,E2 -6779.741} C_VEL
LIN {X 0,Y 481.677,Z 52.481,A -85,B 0,C 180,E1 -6782.674,E2 -6782.674} C_VEL
LIN {X 0,Y 481.646,Z 52.493,A -85,B 0,C 180,E1 -6785.709,E2 -6785.709} C_VEL
LIN {X 0,Y 481.675,Z 52.482,A -85,B 0,C 180,E1 -6788.859,E2 -6788.859} C_VEL
LIN {X 0,Y 481.657,Z 52.486,A -85,B 0,C 180,E1 -6791.913,E2 -6791.913} C_VEL
LIN {X 0,Y 481.659,Z 52.483,A -85,B 0,C 180,E1 -6794.458,E2 -6794.458} C_VEL
LIN {X 0,Y 481.651,Z 52.485,A -85,B 0,C 180,E1 -6797.839,E2 -6797.839} C_VEL
LIN {X 0,Y 481.684,Z 52.482,A -85,B 0,C 180,E1 -6800.651,E2 -6800.651} C_VEL
LIN {X 0,Y 481.631,Z 52.491,A -85,B 0,C 180,E1 -6803.376,E2 -6803.376} C_VEL
LIN {X 0,Y 481.713,Z 52.477,A -85,B 0,C 180,E1 -6806.33,E2 -6806.33} C_VEL
LIN {X 0,Y 481.654,Z 52.485,A -85,B 0,C 180,E1 -6809.417,E2 -6809.417} C_VEL
LIN {X 0,Y 481.703,Z 52.479,A -85,B 0,C 180,E1 -6812.168,E2 -6812.168} C_VEL
LIN {X 0,Y 481.722,Z 52.479,A -85,B 0,C 180,E1 -6814.97,E2 -6814.97} C_VEL
LIN {X 0,Y 481.653,Z 52.484,A -85,B 0,C 180,E1 -6817.705,E2 -6817.705} C_VEL
LIN {X 0,Y 481.708,Z 52.484,A -85,B 0,C 180,E1 -6820.393,E2 -6820.393} C_VEL
LIN {X 0,Y 481.691,Z 52.48,A -85,B 0,C 180,E1 -6823.034,E2 -6823.034} C_VEL
LIN {X 0,Y 481.692,Z 52.48,A -85,B 0,C 180,E1 -6825.639,E2 -6825.639} C_VEL
LIN {X 0,Y 481.754,Z 52.479,A -85,B 0,C 180,E1 -6828.215,E2 -6828.215} C_VEL
LIN {X 0,Y 481.764,Z 52.472,A -85,B 0,C 180,E1 -6831.611,E2 -6831.611} C_VEL
LIN {X 0,Y 481.812,Z 52.47,A -85,B 0,C 180,E1 -6834.139,E2 -6834.139} C_VEL
LIN {X 0,Y 481.928,Z 52.453,A -85,B 0,C 180,E1 -6837.492,E2 -6837.492} C_VEL
LIN {X 0,Y 481.888,Z 52.454,A -85,B 0,C 180,E1 -6840.835,E2 -6840.835} C_VEL
LIN {X 0,Y 481.928,Z 52.45,A -85,B 0,C 180,E1 -6842.507,E2 -6842.507} C_VEL
LIN {X 0,Y 481.808,Z 52.469,A -85,B 0,C 180,E1 -6845.86,E2 -6845.86} C_VEL
LIN {X 0,Y 481.743,Z 52.473,A -85,B 0,C 180,E1 -6848.389,E2 -6848.389} C_VEL
LIN {X 0,Y 481.753,Z 52.474,A -85,B 0,C 180,E1 -6851.785,E2 -6851.785} C_VEL
LIN {X 0,Y 481.745,Z 52.48,A -85,B 0,C 180,E1 -6855.224,E2 -6855.224} C_VEL
LIN {X 0,Y 481.71,Z 52.48,A -85,B 0,C 180,E1 -6858.722,E2 -6858.722} C_VEL
LIN {X 0,Y 481.647,Z 52.488,A -85,B 0,C 180,E1 -6861.395,E2 -6861.395} C_VEL
LIN {X 0,Y 481.673,Z 52.481,A -85,B 0,C 180,E1 -6864.113,E2 -6864.113} C_VEL
LIN {X 0,Y 481.715,Z 52.48,A -85,B 0,C 180,E1 -6867.131,E2 -6867.131} C_VEL
LIN {X 0,Y 481.68,Z 52.48,A -85,B 0,C 180,E1 -6869.741,E2 -6869.741} C_VEL
LIN {X 0,Y 481.674,Z 52.489,A -85,B 0,C 180,E1 -6872.674,E2 -6872.674} C_VEL
LIN {X 0,Y 481.638,Z 52.486,A -85,B 0,C 180,E1 -6875.709,E2 -6875.709} C_VEL
LIN {X 0,Y 481.672,Z 52.484,A -85,B 0,C 180,E1 -6878.859,E2 -6878.859} C_VEL
LIN {X 0,Y 481.654,Z 52.487,A -85,B 0,C 180,E1 -6881.913,E2 -6881.913} C_VEL
LIN {X 0,Y 481.656,Z 52.488,A -85,B 0,C 180,E1 -6884.458,E2 -6884.458} C_VEL
LIN {X 0,Y 481.649,Z 52.489,A -85,B 0,C 180,E1 -6887.839,E2 -6887.839} C_VEL
LIN {X 0,Y 481.682,Z 52.481,A -85,B 0,C 180,E1 -6890.651,E2 -6890.651} C_VEL
LIN {X 0,Y 481.629,Z 52.488,A -85,B 0,C 180,E1 -6893.376,E2 -6893.376} C_VEL
LIN {X 0,Y 481.712,Z 52.478,A -85,B 0,C 180,E1 -6896.33,E2 -6896.33} C_VEL
LIN {X 0,Y 481.652,Z 52.488,A -85,B 0,C 180,E1 -6899.418,E2 -6899.418} C_VEL
LIN {X 0,Y 481.702,Z 52.485,A -85,B 0,C 180,E1 -6902.168,E2 -6902.168} C_VEL
LIN {X 0,Y 481.763,Z 52.577,A -85,B 0,C 180,E1 -6903.697,E2 -6903.697} C_VEL
LIN {X 0,Y 483.739,Z 63.295,A -85,B 0,C 180,E1 -6905.539,E2 -6905.539} C_VEL
LIN {X 0,Y 483.18,Z 82.26,A -85,B 0,C 180,E1 -6908.576,E2 -6908.576} C_VEL
LIN {X 0,Y 482.471,Z 103.753,A -85,B 0,C 180,E1 -6911.968,E2 -6911.968} C_VEL
LIN {X 0,Y 482.145,Z 113.701,A -85,B 0,C 180,E1 -6913.525,E2 -6913.525} C_VEL
LIN {X 0,Y 484.675,Z 132.937,A -85,B 0,C 180,E1 -6913.903,E2 -6913.903} C_VEL
LIN {X 0,Y 484.107,Z 222.598,A -85,B 0,C 180,E1 -6915.255,E2 -6915.255} C_VEL
LIN {X 0,Y 483.75,Z 235.883,A -85,B 0,C 180,E1 -6915.62,E2 -6915.62} C_VEL
LIN {X 0,Y 483.342,Z 248.077,A -85,B 0,C 180,E1 -6916.118,E2 -6916.118} C_VEL
LIN {X 0,Y 482.953,Z 259.581,A -85,B 0,C 180,E1 -6916.75,E2 -6916.75} C_VEL
LIN {X 0,Y 482.466,Z 271.147,A -85,B 0,C 180,E1 -6917.573,E2 -6917.573} C_VEL
LIN {X 0,Y 482.051,Z 281.984,A -85,B 0,C 180,E1 -6918.542,E2 -6918.542} C_VEL
LIN {X 0,Y 481.678,Z 290.647,A -85,B 0,C 180,E1 -6919.491,E2 -6919.491} C_VEL
LIN {X 0,Y 481.392,Z 298.637,A -85,B 0,C 180,E1 -6920.546,E2 -6920.546} C_VEL
LIN {X 0,Y 481.149,Z 306.448,A -85,B 0,C 180,E1 -6921.812,E2 -6921.812} C_VEL
LIN {X 0,Y 480.959,Z 313.621,A -85,B 0,C 180,E1 -6923.287,E2 -6923.287} C_VEL
LIN {X 0,Y 480.907,Z 318.401,A -85,B 0,C 180,E1 -6924.549,E2 -6924.549} C_VEL
LIN {X 0,Y 480.847,Z 322.051,A -85,B 0,C 180,E1 -6925.809,E2 -6925.809} C_VEL
LIN {X 0,Y 480.918,Z 323.941,A -85,B 0,C 180,E1 -6926.649,E2 -6926.649} C_VEL
LIN {X 0,Y 480.878,Z 325.354,A -85,B 0,C 180,E1 -6927.487,E2 -6927.487} C_VEL
LIN {X 0,Y 480.83,Z 326.358,A -85,B 0,C 180,E1 -6928.325,E2 -6928.325} C_VEL
LIN {X 0,Y 480.774,Z 327.192,A -85,B 0,C 180,E1 -6930,E2 -6930} C_VEL
LIN {X 0,Y 480.83,Z 326.371,A -85,B 0,C 180,E1 -6931.675,E2 -6931.675} C_VEL
LIN {X 0,Y 480.878,Z 325.371,A -85,B 0,C 180,E1 -6932.513,E2 -6932.513} C_VEL
LIN {X 0,Y 480.918,Z 323.971,A -85,B 0,C 180,E1 -6933.351,E2 -6933.351} C_VEL
LIN {X 0,Y 480.838,Z 321.014,A -85,B 0,C 180,E1 -6934.611,E2 -6934.611} C_VEL
LIN {X 0,Y 480.876,Z 317.022,A -85,B 0,C 180,E1 -6935.872,E2 -6935.872} C_VEL
LIN {X 0,Y 481.032,Z 310.9,A -85,B 0,C 180,E1 -6937.344,E2 -6937.344} C_VEL
LIN {X 0,Y 481.226,Z 304.212,A -85,B 0,C 180,E1 -6938.609,E2 -6938.609} C_VEL
LIN {X 0,Y 481.476,Z 295.92,A -85,B 0,C 180,E1 -6939.875,E2 -6939.875} C_VEL
LIN {X 0,Y 481.918,Z 287.454,A -85,B 0,C 180,E1 -6940.928,E2 -6940.928} C_VEL
LIN {X 0,Y 482.33,Z 277.28,A -85,B 0,C 180,E1 -6941.959,E2 -6941.959} C_VEL
LIN {X 0,Y 482.71,Z 266.995,A -85,B 0,C 180,E1 -6942.806,E2 -6942.806} C_VEL
LIN {X 0,Y 483.177,Z 255.456,A -85,B 0,C 180,E1 -6943.564,E2 -6943.564} C_VEL
LIN {X 0,Y 483.655,Z 242.812,A -85,B 0,C 180,E1 -6944.194,E2 -6944.194} C_VEL
LIN {X 0,Y 484.087,Z 229.29,A -85,B 0,C 180,E1 -6944.664,E2 -6944.664} C_VEL
LIN {X 0,Y 484.38,Z 215.746,A -85,B 0,C 180,E1 -6944.951,E2 -6944.951} C_VEL
LIN {X 0,Y 484.755,Z 131.311,A -85,B 0,C 180,E1 -6946.224,E2 -6946.224} C_VEL
LIN {X 0,Y 482.204,Z 113.46,A -85,B 0,C 180,E1 -6946.593,E2 -6946.593} C_VEL
LIN {X 0,Y 482.897,Z 93.41,A -85,B 0,C 180,E1 -6949.778,E2 -6949.778} C_VEL
LIN {X 0,Y 483.535,Z 75.612,A -85,B 0,C 180,E1 -6952.654,E2 -6952.654} C_VEL
LIN {X 0,Y 484.032,Z 64.666,A -85,B 0,C 180,E1 -6954.444,E2 -6954.444} C_VEL
LIN {X 0,Y 482.576,Z 56.428,A -85,B 0,C 180,E1 -6955.906,E2 -6955.906} C_VEL
LIN {X 0,Y 481.773,Z 52.475,A -85,B 0,C 180,E1 -6956.652,E2 -6956.652} C_VEL
LIN {X 0,Y 481.679,Z 52.487,A -85,B 0,C 180,E1 -6959.741,E2 -6959.741} C_VEL
LIN {X 0,Y 481.67,Z 52.487,A -85,B 0,C 180,E1 -6962.674,E2 -6962.674} C_VEL
LIN {X 0,Y 481.642,Z 52.488,A -85,B 0,C 180,E1 -6965.709,E2 -6965.709} C_VEL
LIN {X 0,Y 481.67,Z 52.483,A -85,B 0,C 180,E1 -6968.859,E2 -6968.859} C_VEL
LIN {X 0,Y 481.651,Z 52.49,A -85,B 0,C 180,E1 -6971.912,E2 -6971.912} C_VEL
LIN {X 0,Y 481.653,Z 52.483,A -85,B 0,C 180,E1 -6974.458,E2 -6974.458} C_VEL
LIN {X 0,Y 481.647,Z 52.489,A -85,B 0,C 180,E1 -6977.839,E2 -6977.839} C_VEL
LIN {X 0,Y 481.713,Z 52.477,A -85,B 0,C 180,E1 -6980.646,E2 -6980.646} C_VEL
LIN {X 0,Y 481.641,Z 52.486,A -85,B 0,C 180,E1 -6984.291,E2 -6984.291} C_VEL
LIN {X 0,Y 481.67,Z 52.488,A -85,B 0,C 180,E1 -6987.326,E2 -6987.326} C_VEL
LIN {X 0,Y 481.677,Z 52.481,A -85,B 0,C 180,E1 -6990.259,E2 -6990.259} C_VEL
LIN {X 0,Y 481.743,Z 52.475,A -85,B 0,C 180,E1 -6993.112,E2 -6993.112} C_VEL
LIN {X 0,Y 481.675,Z 52.482,A -85,B 0,C 180,E1 -6995.887,E2 -6995.887} C_VEL
LIN {X 0,Y 481.7,Z 52.481,A -85,B 0,C 180,E1 -6999.027,E2 -6999.027} C_VEL
LIN {X 0,Y 481.705,Z 52.479,A -85,B 0,C 180,E1 -7002.158,E2 -7002.158} C_VEL
LIN {X 0,Y 481.74,Z 52.476,A -85,B 0,C 180,E1 -7004.776,E2 -7004.776} C_VEL
LIN {X 0,Y 481.749,Z 52.475,A -85,B 0,C 180,E1 -7008.215,E2 -7008.215} C_VEL
LIN {X 0,Y 481.761,Z 52.472,A -85,B 0,C 180,E1 -7011.612,E2 -7011.612} C_VEL
LIN {X 0,Y 481.808,Z 52.471,A -85,B 0,C 180,E1 -7014.14,E2 -7014.14} C_VEL
LIN {X 0,Y 481.924,Z 52.451,A -85,B 0,C 180,E1 -7017.493,E2 -7017.493} C_VEL
LIN {X 0,Y 481.937,Z 52.454,A -85,B 0,C 180,E1 -7020,E2 -7020} C_VEL
LIN {X 0,Y 481.924,Z 52.446,A -85,B 0,C 180,E1 -7022.508,E2 -7022.508} C_VEL
LIN {X 0,Y 481.804,Z 52.468,A -85,B 0,C 180,E1 -7025.861,E2 -7025.861} C_VEL
LIN {X 0,Y 481.738,Z 52.469,A -85,B 0,C 180,E1 -7028.389,E2 -7028.389} C_VEL
LIN {X 0,Y 481.749,Z 52.472,A -85,B 0,C 180,E1 -7031.785,E2 -7031.785} C_VEL
LIN {X 0,Y 481.74,Z 52.48,A -85,B 0,C 180,E1 -7035.225,E2 -7035.225} C_VEL
LIN {X 0,Y 481.706,Z 52.48,A -85,B 0,C 180,E1 -7038.722,E2 -7038.722} C_VEL
LIN {X 0,Y 481.644,Z 52.483,A -85,B 0,C 180,E1 -7041.395,E2 -7041.395} C_VEL
LIN {X 0,Y 481.661,Z 52.485,A -85,B 0,C 180,E1 -7044.114,E2 -7044.114} C_VEL
LIN {X 0,Y 481.693,Z 52.482,A -85,B 0,C 180,E1 -7047.127,E2 -7047.127} C_VEL
LIN {X 0,Y 481.672,Z 52.481,A -85,B 0,C 180,E1 -7049.742,E2 -7049.742} C_VEL
LIN {X 0,Y 481.669,Z 52.487,A -85,B 0,C 180,E1 -7052.675,E2 -7052.675} C_VEL
LIN {X 0,Y 481.63,Z 52.487,A -85,B 0,C 180,E1 -7055.711,E2 -7055.711} C_VEL
LIN {X 0,Y 481.665,Z 52.486,A -85,B 0,C 180,E1 -7058.86,E2 -7058.86} C_VEL
LIN {X 0,Y 481.628,Z 52.494,A -85,B 0,C 180,E1 -7062.163,E2 -7062.163} C_VEL
LIN {X 0,Y 481.654,Z 52.487,A -85,B 0,C 180,E1 -7065.543,E2 -7065.543} C_VEL
LIN {X 0,Y 481.632,Z 52.489,A -85,B 0,C 180,E1 -7068.956,E2 -7068.956} C_VEL
LIN {X 0,Y 481.635,Z 52.492,A -85,B 0,C 180,E1 -7071.997,E2 -7071.997} C_VEL
LIN {X 0,Y 481.684,Z 52.488,A -85,B 0,C 180,E1 -7075.318,E2 -7075.318} C_VEL
LIN {X 0,Y 481.735,Z 52.602,A -85,B 0,C 180,E1 -7076.615,E2 -7076.615} C_VEL
LIN {X 0,Y 482.741,Z 58.764,A -85,B 0,C 180,E1 -7078.024,E2 -7078.024} C_VEL
LIN {X 0,Y 482.665,Z 65.734,A -85,B 0,C 180,E1 -7079.49,E2 -7079.49} C_VEL
LIN {X 0,Y 485.259,Z 77.781,A -85,B 0,C 180,E1 -7079.777,E2 -7079.777} C_VEL
LIN {X 0,Y 484.949,Z 122.395,A -85,B 0,C 180,E1 -7080.448,E2 -7080.448} C_VEL
LIN {X 0,Y 484.275,Z 128.24,A -85,B 0,C 180,E1 -7080.512,E2 -7080.512} C_VEL
LIN {X 0,Y 478.52,Z 147.227,A -85,B 0,C 180,E1 -7080.592,E2 -7080.592} C_VEL
LIN {X 0,Y 477.861,Z 153.071,A -85,B 0,C 180,E1 -7080.658,E2 -7080.658} C_VEL
LIN {X 0,Y 477.689,Z 174.112,A -85,B 0,C 180,E1 -7081.015,E2 -7081.015} C_VEL
LIN {X 0,Y 477.474,Z 186.702,A -85,B 0,C 180,E1 -7081.391,E2 -7081.391} C_VEL
LIN {X 0,Y 477.174,Z 199.307,A -85,B 0,C 180,E1 -7081.945,E2 -7081.945} C_VEL
LIN {X 0,Y 476.731,Z 210.743,A -85,B 0,C 180,E1 -7082.621,E2 -7082.621} C_VEL
LIN {X 0,Y 476.203,Z 222.167,A -85,B 0,C 180,E1 -7083.485,E2 -7083.485} C_VEL
LIN {X 0,Y 475.748,Z 232.954,A -85,B 0,C 180,E1 -7084.517,E2 -7084.517} C_VEL
LIN {X 0,Y 475.297,Z 241.628,A -85,B 0,C 180,E1 -7085.543,E2 -7085.543} C_VEL
LIN {X 0,Y 474.909,Z 249.43,A -85,B 0,C 180,E1 -7086.663,E2 -7086.663} C_VEL
LIN {X 0,Y 474.517,Z 257.194,A -85,B 0,C 180,E1 -7088.04,E2 -7088.04} C_VEL
LIN {X 0,Y 474.322,Z 262.296,A -85,B 0,C 180,E1 -7089.17,E2 -7089.17} C_VEL
LIN {X 0,Y 474.133,Z 267.168,A -85,B 0,C 180,E1 -7090.518,E2 -7090.518} C_VEL
LIN {X 0,Y 473.94,Z 270.816,A -85,B 0,C 180,E1 -7091.856,E2 -7091.856} C_VEL
LIN {X 0,Y 473.815,Z 272.622,A -85,B 0,C 180,E1 -7092.744,E2 -7092.744} C_VEL
LIN {X 0,Y 473.801,Z 273.968,A -85,B 0,C 180,E1 -7093.631,E2 -7093.631} C_VEL
LIN {X 0,Y 473.763,Z 275.002,A -85,B 0,C 180,E1 -7094.633,E2 -7094.633} C_VEL
LIN {X 0,Y 473.739,Z 275.449,A -85,B 0,C 180,E1 -7096.269,E2 -7096.269} C_VEL
LIN {X 0,Y 473.75,Z 275.108,A -85,B 0,C 180,E1 -7097.143,E2 -7097.143} C_VEL
LIN {X 0,Y 473.839,Z 274.12,A -85,B 0,C 180,E1 -7098.216,E2 -7098.216} C_VEL
LIN {X 0,Y 473.899,Z 271.58,A -85,B 0,C 180,E1 -7099.749,E2 -7099.749} C_VEL
LIN {X 0,Y 474.007,Z 268.361,A -85,B 0,C 180,E1 -7101.044,E2 -7101.044} C_VEL
LIN {X 0,Y 474.175,Z 264.072,A -85,B 0,C 180,E1 -7102.335,E2 -7102.335} C_VEL
LIN {X 0,Y 474.387,Z 257.603,A -85,B 0,C 180,E1 -7103.834,E2 -7103.834} C_VEL
LIN {X 0,Y 474.724,Z 250.492,A -85,B 0,C 180,E1 -7105.117,E2 -7105.117} C_VEL
LIN {X 0,Y 475.099,Z 241.673,A -85,B 0,C 180,E1 -7106.396,E2 -7106.396} C_VEL
LIN {X 0,Y 475.549,Z 232.625,A -85,B 0,C 180,E1 -7107.459,E2 -7107.459} C_VEL
LIN {X 0,Y 475.962,Z 222.626,A -85,B 0,C 180,E1 -7108.414,E2 -7108.414} C_VEL
LIN {X 0,Y 476.451,Z 211.514,A -85,B 0,C 180,E1 -7109.261,E2 -7109.261} C_VEL
LIN {X 0,Y 476.842,Z 199.106,A -85,B 0,C 180,E1 -7110,E2 -7110} C_VEL
LIN {X 0,Y 477.069,Z 186.431,A -85,B 0,C 180,E1 -7110.554,E2 -7110.554} C_VEL
LIN {X 0,Y 477.37,Z 172.804,A -85,B 0,C 180,E1 -7110.949,E2 -7110.949} C_VEL
LIN {X 0,Y 477.877,Z 108.251,A -85,B 0,C 180,E1 -7111.949,E2 -7111.949} C_VEL
LIN {X 0,Y 477.927,Z 77.705,A -85,B 0,C 180,E1 -7112.417,E2 -7112.417} C_VEL
LIN {X 0,Y 475.434,Z 65.47,A -85,B 0,C 180,E1 -7112.701,E2 -7112.701} C_VEL
LIN {X 0,Y 475.493,Z 58.326,A -85,B 0,C 180,E1 -7114.238,E2 -7114.238} C_VEL
LIN {X 0,Y 474.804,Z 53.343,A -85,B 0,C 180,E1 -7115.362,E2 -7115.362} C_VEL
LIN {X 0,Y 474.801,Z 53.34,A -85,B 0,C 180,E1 -7117.656,E2 -7117.656} C_VEL
LIN {X 0,Y 474.682,Z 53.354,A -85,B 0,C 180,E1 -7121.097,E2 -7121.097} C_VEL
LIN {X 0,Y 474.646,Z 53.357,A -85,B 0,C 180,E1 -7123.704,E2 -7123.704} C_VEL
LIN {X 0,Y 474.645,Z 53.364,A -85,B 0,C 180,E1 -7126.34,E2 -7126.34} C_VEL
LIN {X 0,Y 474.669,Z 53.354,A -85,B 0,C 180,E1 -7129.01,E2 -7129.01} C_VEL
LIN {X 0,Y 474.594,Z 53.365,A -85,B 0,C 180,E1 -7131.729,E2 -7131.729} C_VEL
LIN {X 0,Y 474.646,Z 53.359,A -85,B 0,C 180,E1 -7134.494,E2 -7134.494} C_VEL
LIN {X 0,Y 474.686,Z 53.353,A -85,B 0,C 180,E1 -7137.334,E2 -7137.334} C_VEL
LIN {X 0,Y 474.609,Z 53.361,A -85,B 0,C 180,E1 -7140.81,E2 -7140.81} C_VEL
LIN {X 0,Y 474.643,Z 53.362,A -85,B 0,C 180,E1 -7143.984,E2 -7143.984} C_VEL
LIN {X 0,Y 474.579,Z 53.365,A -85,B 0,C 180,E1 -7146.899,E2 -7146.899} C_VEL
LIN {X 0,Y 474.632,Z 53.365,A -85,B 0,C 180,E1 -7149.647,E2 -7149.647} C_VEL
LIN {X 0,Y 474.619,Z 53.362,A -85,B 0,C 180,E1 -7152.934,E2 -7152.934} C_VEL
LIN {X 0,Y 474.61,Z 53.363,A -85,B 0,C 180,E1 -7155.895,E2 -7155.895} C_VEL
LIN {X 0,Y 474.631,Z 53.364,A -85,B 0,C 180,E1 -7159.041,E2 -7159.041} C_VEL
LIN {X 0,Y 474.614,Z 53.362,A -85,B 0,C 180,E1 -7161.704,E2 -7161.704} C_VEL
LIN {X 0,Y 474.629,Z 53.363,A -85,B 0,C 180,E1 -7164.726,E2 -7164.726} C_VEL
LIN {X 0,Y 474.639,Z 53.358,A -85,B 0,C 180,E1 -7167.788,E2 -7167.788} C_VEL
LIN {X 0,Y 474.628,Z 53.366,A -85,B 0,C 180,E1 -7170.884,E2 -7170.884} C_VEL
LIN {X 0,Y 474.664,Z 53.354,A -85,B 0,C 180,E1 -7173.628,E2 -7173.628} C_VEL
LIN {X 0,Y 474.639,Z 53.365,A -85,B 0,C 180,E1 -7176.641,E2 -7176.641} C_VEL
LIN {X 0,Y 474.658,Z 53.358,A -85,B 0,C 180,E1 -7180.089,E2 -7180.089} C_VEL
LIN {X 0,Y 474.651,Z 53.359,A -85,B 0,C 180,E1 -7182.774,E2 -7182.774} C_VEL
LIN {X 0,Y 474.651,Z 53.356,A -85,B 0,C 180,E1 -7185.421,E2 -7185.421} C_VEL
LIN {X 0,Y 474.707,Z 53.355,A -85,B 0,C 180,E1 -7188.037,E2 -7188.037} C_VEL
LIN {X 0,Y 474.729,Z 53.348,A -85,B 0,C 180,E1 -7191.486,E2 -7191.486} C_VEL
LIN {X 0,Y 474.775,Z 53.348,A -85,B 0,C 180,E1 -7194.052,E2 -7194.052} C_VEL
LIN {X 0,Y 474.895,Z 53.328,A -85,B 0,C 180,E1 -7197.455,E2 -7197.455} C_VEL
LIN {X 0,Y 474.913,Z 53.329,A -85,B 0,C 180,E1 -7200,E2 -7200} C_VEL
LIN {X 0,Y 474.894,Z 53.326,A -85,B 0,C 180,E1 -7202.544,E2 -7202.544} C_VEL
LIN {X 0,Y 474.771,Z 53.344,A -85,B 0,C 180,E1 -7205.948,E2 -7205.948} C_VEL
LIN {X 0,Y 474.714,Z 53.348,A -85,B 0,C 180,E1 -7208.514,E2 -7208.514} C_VEL
LIN {X 0,Y 474.706,Z 53.35,A -85,B 0,C 180,E1 -7211.962,E2 -7211.962} C_VEL
LIN {X 0,Y 474.702,Z 53.355,A -85,B 0,C 180,E1 -7215.455,E2 -7215.455} C_VEL
LIN {X 0,Y 474.665,Z 53.361,A -85,B 0,C 180,E1 -7219.01,E2 -7219.01} C_VEL
LIN {X 0,Y 474.59,Z 53.364,A -85,B 0,C 180,E1 -7221.729,E2 -7221.729} C_VEL
LIN {X 0,Y 474.652,Z 53.358,A -85,B 0,C 180,E1 -7224.493,E2 -7224.493} C_VEL
LIN {X 0,Y 474.675,Z 53.355,A -85,B 0,C 180,E1 -7227.332,E2 -7227.332} C_VEL
LIN {X 0,Y 474.607,Z 53.364,A -85,B 0,C 180,E1 -7230.23,E2 -7230.23} C_VEL
LIN {X 0,Y 474.645,Z 53.358,A -85,B 0,C 180,E1 -7233.22,E2 -7233.22} C_VEL
LIN {X 0,Y 474.591,Z 53.369,A -85,B 0,C 180,E1 -7236.323,E2 -7236.323} C_VEL
LIN {X 0,Y 474.62,Z 53.36,A -85,B 0,C 180,E1 -7239.646,E2 -7239.646} C_VEL
LIN {X 0,Y 474.626,Z 53.366,A -85,B 0,C 180,E1 -7242.237,E2 -7242.237} C_VEL
LIN {X 0,Y 474.618,Z 53.36,A -85,B 0,C 180,E1 -7245.298,E2 -7245.298} C_VEL
LIN {X 0,Y 474.622,Z 53.366,A -85,B 0,C 180,E1 -7248.214,E2 -7248.214} C_VEL
LIN {X 0,Y 474.646,Z 53.359,A -85,B 0,C 180,E1 -7250.454,E2 -7250.454} C_VEL
LIN {X 0,Y 474.591,Z 53.368,A -85,B 0,C 180,E1 -7253.676,E2 -7253.676} C_VEL
LIN {X 0,Y 474.645,Z 53.357,A -85,B 0,C 180,E1 -7256.78,E2 -7256.78} C_VEL
LIN {X 0,Y 474.607,Z 53.369,A -85,B 0,C 180,E1 -7259.77,E2 -7259.77} C_VEL
LIN {X 0,Y 474.726,Z 53.355,A -85,B 0,C 180,E1 -7263.158,E2 -7263.158} C_VEL
LIN {X 0,Y 474.694,Z 53.398,A -85,B 0,C 180,E1 -7263.512,E2 -7263.512} C_VEL
LIN {X 0,Y 476.735,Z 64.144,A -85,B 0,C 180,E1 -7265.388,E2 -7265.388} C_VEL
LIN {X 0,Y 476.35,Z 76.745,A -85,B 0,C 180,E1 -7267.443,E2 -7267.443} C_VEL
LIN {X 0,Y 475.771,Z 93.496,A -85,B 0,C 180,E1 -7270.138,E2 -7270.138} C_VEL
LIN {X 0,Y 475.226,Z 110.162,A -85,B 0,C 180,E1 -7272.796,E2 -7272.796} C_VEL
LIN {X 0,Y 475.155,Z 113.351,A -85,B 0,C 180,E1 -7273.303,E2 -7273.303} C_VEL
LIN {X 0,Y 477.81,Z 134.128,A -85,B 0,C 180,E1 -7273.711,E2 -7273.711} C_VEL
LIN {X 0,Y 477.177,Z 222.435,A -85,B 0,C 180,E1 -7275.063,E2 -7275.063} C_VEL
LIN {X 0,Y 476.826,Z 235.661,A -85,B 0,C 180,E1 -7275.434,E2 -7275.434} C_VEL
LIN {X 0,Y 476.383,Z 248.393,A -85,B 0,C 180,E1 -7275.966,E2 -7275.966} C_VEL
LIN {X 0,Y 475.936,Z 260.51,A -85,B 0,C 180,E1 -7276.66,E2 -7276.66} C_VEL
LIN {X 0,Y 475.448,Z 271.602,A -85,B 0,C 180,E1 -7277.476,E2 -7277.476} C_VEL
LIN {X 0,Y 475.003,Z 282.498,A -85,B 0,C 180,E1 -7278.478,E2 -7278.478} C_VEL
LIN {X 0,Y 474.573,Z 291.853,A -85,B 0,C 180,E1 -7279.548,E2 -7279.548} C_VEL
LIN {X 0,Y 474.219,Z 300.93,A -85,B 0,C 180,E1 -7280.832,E2 -7280.832} C_VEL
LIN {X 0,Y 474.006,Z 308.238,A -85,B 0,C 180,E1 -7282.117,E2 -7282.117} C_VEL
LIN {X 0,Y 473.891,Z 313.174,A -85,B 0,C 180,E1 -7283.186,E2 -7283.186} C_VEL
LIN {X 0,Y 473.817,Z 317.969,A -85,B 0,C 180,E1 -7284.467,E2 -7284.467} C_VEL
LIN {X 0,Y 473.75,Z 321.633,A -85,B 0,C 180,E1 -7285.746,E2 -7285.746} C_VEL
LIN {X 0,Y 473.841,Z 323.531,A -85,B 0,C 180,E1 -7286.598,E2 -7286.598} C_VEL
LIN {X 0,Y 473.793,Z 324.953,A -85,B 0,C 180,E1 -7287.449,E2 -7287.449} C_VEL
LIN {X 0,Y 473.764,Z 325.963,A -85,B 0,C 180,E1 -7288.3,E2 -7288.3} C_VEL
LIN {X 0,Y 473.698,Z 326.807,A -85,B 0,C 180,E1 -7290,E2 -7290} C_VEL
LIN {X 0,Y 473.708,Z 326.603,A -85,B 0,C 180,E1 -7290.85,E2 -7290.85} C_VEL
LIN {X 0,Y 473.764,Z 325.999,A -85,B 0,C 180,E1 -7291.7,E2 -7291.7} C_VEL
LIN {X 0,Y 473.792,Z 325.003,A -85,B 0,C 180,E1 -7292.55,E2 -7292.55} C_VEL
LIN {X 0,Y 473.841,Z 323.609,A -85,B 0,C 180,E1 -7293.401,E2 -7293.401} C_VEL
LIN {X 0,Y 473.76,Z 320.661,A -85,B 0,C 180,E1 -7294.68,E2 -7294.68} C_VEL
LIN {X 0,Y 473.787,Z 316.681,A -85,B 0,C 180,E1 -7295.96,E2 -7295.96} C_VEL
LIN {X 0,Y 473.97,Z 310.581,A -85,B 0,C 180,E1 -7297.454,E2 -7297.454} C_VEL
LIN {X 0,Y 474.135,Z 303.912,A -85,B 0,C 180,E1 -7298.739,E2 -7298.739} C_VEL
LIN {X 0,Y 474.423,Z 295.65,A -85,B 0,C 180,E1 -7300.024,E2 -7300.024} C_VEL
LIN {X 0,Y 474.909,Z 287.22,A -85,B 0,C 180,E1 -7301.091,E2 -7301.091} C_VEL
LIN {X 0,Y 475.34,Z 277.3,A -85,B 0,C 180,E1 -7302.12,E2 -7302.12} C_VEL
LIN {X 0,Y 475.786,Z 266.584,A -85,B 0,C 180,E1 -7303.018,E2 -7303.018} C_VEL
LIN {X 0,Y 476.277,Z 255.398,A -85,B 0,C 180,E1 -7303.765,E2 -7303.765} C_VEL
LIN {X 0,Y 476.79,Z 242.91,A -85,B 0,C 180,E1 -7304.403,E2 -7304.403} C_VEL
LIN {X 0,Y 477.242,Z 229.589,A -85,B 0,C 180,E1 -7304.879,E2 -7304.879} C_VEL
LIN {X 0,Y 477.558,Z 216.598,A -85,B 0,C 180,E1 -7305.169,E2 -7305.169} C_VEL
LIN {X 0,Y 477.98,Z 132.092,A -85,B 0,C 180,E1 -7306.464,E2 -7306.464} C_VEL
LIN {X 0,Y 475.226,Z 112.904,A -85,B 0,C 180,E1 -7306.892,E2 -7306.892} C_VEL
LIN {X 0,Y 475.984,Z 93.204,A -85,B 0,C 180,E1 -7310.077,E2 -7310.077} C_VEL
LIN {X 0,Y 476.804,Z 72.699,A -85,B 0,C 180,E1 -7313.451,E2 -7313.451} C_VEL
LIN {X 0,Y 477.124,Z 65.87,A -85,B 0,C 180,E1 -7314.589,E2 -7314.589} C_VEL
LIN {X 0,Y 475.365,Z 56.286,A -85,B 0,C 180,E1 -7316.329,E2 -7316.329} C_VEL
LIN {X 0,Y 474.705,Z 53.357,A -85,B 0,C 180,E1 -7316.902,E2 -7316.902} C_VEL
LIN {X 0,Y 474.605,Z 53.37,A -85,B 0,C 180,E1 -7320.23,E2 -7320.23} C_VEL
LIN {X 0,Y 474.633,Z 53.362,A -85,B 0,C 180,E1 -7323.22,E2 -7323.22} C_VEL
LIN {X 0,Y 474.593,Z 53.369,A -85,B 0,C 180,E1 -7326.323,E2 -7326.323} C_VEL
LIN {X 0,Y 474.626,Z 53.366,A -85,B 0,C 180,E1 -7329.647,E2 -7329.647} C_VEL
LIN {X 0,Y 474.613,Z 53.363,A -85,B 0,C 180,E1 -7332.934,E2 -7332.934} C_VEL
LIN {X 0,Y 474.604,Z 53.361,A -85,B 0,C 180,E1 -7335.894,E2 -7335.894} C_VEL
LIN {X 0,Y 474.639,Z 53.361,A -85,B 0,C 180,E1 -7339.039,E2 -7339.039} C_VEL
LIN {X 0,Y 474.615,Z 53.362,A -85,B 0,C 180,E1 -7341.703,E2 -7341.703} C_VEL
LIN {X 0,Y 474.628,Z 53.362,A -85,B 0,C 180,E1 -7344.726,E2 -7344.726} C_VEL
LIN {X 0,Y 474.634,Z 53.36,A -85,B 0,C 180,E1 -7347.788,E2 -7347.788} C_VEL
LIN {X 0,Y 474.622,Z 53.366,A -85,B 0,C 180,E1 -7350.884,E2 -7350.884} C_VEL
LIN {X 0,Y 474.658,Z 53.354,A -85,B 0,C 180,E1 -7353.628,E2 -7353.628} C_VEL
LIN {X 0,Y 474.634,Z 53.363,A -85,B 0,C 180,E1 -7356.641,E2 -7356.641} C_VEL
LIN {X 0,Y 474.654,Z 53.358,A -85,B 0,C 180,E1 -7360.09,E2 -7360.09} C_VEL
LIN {X 0,Y 474.648,Z 53.36,A -85,B 0,C 180,E1 -7362.774,E2 -7362.774} C_VEL
LIN {X 0,Y 474.645,Z 53.357,A -85,B 0,C 180,E1 -7365.421,E2 -7365.421} C_VEL
LIN {X 0,Y 474.702,Z 53.35,A -85,B 0,C 180,E1 -7368.038,E2 -7368.038} C_VEL
LIN {X 0,Y 474.726,Z 53.347,A -85,B 0,C 180,E1 -7371.487,E2 -7371.487} C_VEL
LIN {X 0,Y 474.77,Z 53.348,A -85,B 0,C 180,E1 -7374.052,E2 -7374.052} C_VEL
LIN {X 0,Y 474.891,Z 53.327,A -85,B 0,C 180,E1 -7377.456,E2 -7377.456} C_VEL
LIN {X 0,Y 474.908,Z 53.329,A -85,B 0,C 180,E1 -7380,E2 -7380} C_VEL
LIN {X 0,Y 474.89,Z 53.322,A -85,B 0,C 180,E1 -7382.545,E2 -7382.545} C_VEL
LIN {X 0,Y 474.767,Z 53.344,A -85,B 0,C 180,E1 -7385.948,E2 -7385.948} C_VEL
LIN {X 0,Y 474.71,Z 53.345,A -85,B 0,C 180,E1 -7388.514,E2 -7388.514} C_VEL
LIN {X 0,Y 474.702,Z 53.348,A -85,B 0,C 180,E1 -7391.963,E2 -7391.963} C_VEL
LIN {X 0,Y 474.698,Z 53.354,A -85,B 0,C 180,E1 -7395.456,E2 -7395.456} C_VEL
LIN {X 0,Y 474.661,Z 53.362,A -85,B 0,C 180,E1 -7399.011,E2 -7399.011} C_VEL
LIN {X 0,Y 474.586,Z 53.361,A -85,B 0,C 180,E1 -7401.729,E2 -7401.729} C_VEL
LIN {X 0,Y 474.639,Z 53.364,A -85,B 0,C 180,E1 -7404.494,E2 -7404.494} C_VEL
LIN {X 0,Y 474.635,Z 53.36,A -85,B 0,C 180,E1 -7407.324,E2 -7407.324} C_VEL
LIN {X 0,Y 474.602,Z 53.366,A -85,B 0,C 180,E1 -7410.231,E2 -7410.231} C_VEL
LIN {X 0,Y 474.624,Z 53.36,A -85,B 0,C 180,E1 -7413.222,E2 -7413.222} C_VEL
LIN {X 0,Y 474.583,Z 53.373,A -85,B 0,C 180,E1 -7416.325,E2 -7416.325} C_VEL
LIN {X 0,Y 474.621,Z 53.365,A -85,B 0,C 180,E1 -7419.549,E2 -7419.549} C_VEL
LIN {X 0,Y 474.587,Z 53.372,A -85,B 0,C 180,E1 -7422.232,E2 -7422.232} C_VEL
LIN {X 0,Y 474.616,Z 53.362,A -85,B 0,C 180,E1 -7425.298,E2 -7425.298} C_VEL
LIN {X 0,Y 474.604,Z 53.366,A -85,B 0,C 180,E1 -7428.213,E2 -7428.213} C_VEL
LIN {X 0,Y 474.6,Z 53.371,A -85,B 0,C 180,E1 -7431.542,E2 -7431.542} C_VEL
LIN {X 0,Y 474.62,Z 53.366,A -85,B 0,C 180,E1 -7434.726,E2 -7434.726} C_VEL
LIN {X 0,Y 474.676,Z 53.489,A -85,B 0,C 180,E1 -7436.408,E2 -7436.408} C_VEL
LIN {X 0,Y 475.774,Z 59.805,A -85,B 0,C 180,E1 -7437.875,E2 -7437.875} C_VEL
LIN {X 0,Y 475.713,Z 65.996,A -85,B 0,C 180,E1 -7439.211,E2 -7439.211} C_VEL
LIN {X 0,Y 478.553,Z 79.403,A -85,B 0,C 180,E1 -7439.537,E2 -7439.537} C_VEL
LIN {X 0,Y 477.861,Z 153.071,A -85,B 0,C 180,E1 -7440.658,E2 -7440.658} C_VEL
LIN {X 0,Y 477.235,Z 158.921,A -85,B 0,C 180,E1 -7440.723,E2 -7440.723} C_VEL
LIN {X 0,Y 472.047,Z 175.973,A -85,B 0,C 180,E1 -7440.842,E2 -7440.842} C_VEL
LIN {X 0,Y 470.895,Z 181.675,A -85,B 0,C 180,E1 -7440.962,E2 -7440.962} C_VEL
LIN {X 0,Y 470.743,Z 183.575,A -85,B 0,C 180,E1 -7441.021,E2 -7441.021} C_VEL
LIN {X 0,Y 470.471,Z 195.739,A -85,B 0,C 180,E1 -7441.514,E2 -7441.514} C_VEL
LIN {X 0,Y 470.037,Z 207.649,A -85,B 0,C 180,E1 -7442.168,E2 -7442.168} C_VEL
LIN {X 0,Y 469.485,Z 218.767,A -85,B 0,C 180,E1 -7442.955,E2 -7442.955} C_VEL
LIN {X 0,Y 469.028,Z 228.791,A -85,B 0,C 180,E1 -7443.848,E2 -7443.848} C_VEL
LIN {X 0,Y 468.571,Z 238.599,A -85,B 0,C 180,E1 -7444.931,E2 -7444.931} C_VEL
LIN {X 0,Y 468.072,Z 247.135,A -85,B 0,C 180,E1 -7446.084,E2 -7446.084} C_VEL
LIN {X 0,Y 467.655,Z 255.39,A -85,B 0,C 180,E1 -7447.467,E2 -7447.467} C_VEL
LIN {X 0,Y 467.329,Z 261.854,A -85,B 0,C 180,E1 -7448.843,E2 -7448.843} C_VEL
LIN {X 0,Y 467.113,Z 266.906,A -85,B 0,C 180,E1 -7450.213,E2 -7450.213} C_VEL
LIN {X 0,Y 466.888,Z 270.721,A -85,B 0,C 180,E1 -7451.573,E2 -7451.573} C_VEL
LIN {X 0,Y 466.781,Z 272.663,A -85,B 0,C 180,E1 -7452.475,E2 -7452.475} C_VEL
LIN {X 0,Y 466.732,Z 274.103,A -85,B 0,C 180,E1 -7453.376,E2 -7453.376} C_VEL
LIN {X 0,Y 466.699,Z 275.341,A -85,B 0,C 180,E1 -7454.533,E2 -7454.533} C_VEL
LIN {X 0,Y 466.649,Z 275.872,A -85,B 0,C 180,E1 -7456.057,E2 -7456.057} C_VEL
LIN {X 0,Y 466.676,Z 275.6,A -85,B 0,C 180,E1 -7456.945,E2 -7456.945} C_VEL
LIN {X 0,Y 466.765,Z 274.599,A -85,B 0,C 180,E1 -7458.154,E2 -7458.154} C_VEL
LIN {X 0,Y 466.799,Z 272.359,A -85,B 0,C 180,E1 -7459.592,E2 -7459.592} C_VEL
